LIN {X 0,Y 440.779,Z 670.72,A -85,B 0,C 180,E1 8798.14,E2 8798.14} C_VEL
LIN {X 0,Y 437.985,Z 696.597,A -85,B 0,C 180,E1 8801.691,E2 8801.691} C_VEL
LIN {X 0,Y 435.886,Z 717.468,A -85,B 0,C 180,E1 8805.769,E2 8805.769} C_VEL
LIN {X 0,Y 434.77,Z 732.2,A -85,B 0,C 180,E1 8810.004,E2 8810.004} C_VEL
LIN {X 0,Y 434.32,Z 740.921,A -85,B 0,C 180,E1 8814.015,E2 8814.015} C_VEL
LIN {X 0,Y 434.115,Z 745.167,A -85,B 0,C 180,E1 8818.005,E2 8818.005} C_VEL
LIN {X 0,Y 434.245,Z 745.196,A -85,B 0,C 180,E1 8821.989,E2 8821.989} C_VEL
LIN {X 0,Y 434.323,Z 741.018,A -85,B 0,C 180,E1 8825.98,E2 8825.98} C_VEL
LIN {X 0,Y 434.91,Z 730.868,A -85,B 0,C 180,E1 8830.493,E2 8830.493} C_VEL
LIN {X 0,Y 436.273,Z 714.903,A -85,B 0,C 180,E1 8834.818,E2 8834.818} C_VEL
LIN {X 0,Y 438.333,Z 693.903,A -85,B 0,C 180,E1 8838.674,E2 8838.674} C_VEL
LIN {X 0,Y 441.086,Z 667.612,A -85,B 0,C 180,E1 8842.103,E2 8842.103} C_VEL
LIN {X 0,Y 444.082,Z 637.747,A -85,B 0,C 180,E1 8844.863,E2 8844.863} C_VEL
LIN {X 0,Y 446.927,Z 603.336,A -85,B 0,C 180,E1 8847.021,E2 8847.021} C_VEL
LIN {X 0,Y 448.217,Z 571.069,A -85,B 0,C 180,E1 8848.344,E2 8848.344} C_VEL
LIN {X 0,Y 435.993,Z 537.616,A -85,B 0,C 180,E1 8850.23,E2 8850.23} C_VEL
LIN {X 0,Y 432.921,Z 529.66,A -85,B 0,C 180,E1 8850.787,E2 8850.787} C_VEL
LIN {X 0,Y 432.776,Z 529.66,A -85,B 0,C 180,E1 8856.684,E2 8856.684} C_VEL
LIN {X 0,Y 432.689,Z 529.66,A -85,B 0,C 180,E1 8862.916,E2 8862.916} C_VEL
LIN {X 0,Y 432.797,Z 529.66,A -85,B 0,C 180,E1 8868.514,E2 8868.514} C_VEL
LIN {X 0,Y 432.948,Z 530.172,A -85,B 0,C 180,E1 8874.712,E2 8874.712} C_VEL
LIN {X 0,Y 445.086,Z 561.236,A -85,B 0,C 180,E1 8876.436,E2 8876.436} C_VEL
LIN {X 0,Y 450.898,Z 581.785,A -85,B 0,C 180,E1 8877.342,E2 8877.342} C_VEL
LIN {X 0,Y 450.65,Z 585.781,A -85,B 0,C 180,E1 8877.438,E2 8877.438} C_VEL
LIN {X 0,Y 446.315,Z 602.62,A -85,B 0,C 180,E1 8877.748,E2 8877.748} C_VEL
LIN {X 0,Y 441.689,Z 619.155,A -85,B 0,C 180,E1 8878.204,E2 8878.204} C_VEL
LIN {X 0,Y 438.626,Z 656.172,A -85,B 0,C 180,E1 8880.362,E2 8880.362} C_VEL
LIN {X 0,Y 435.196,Z 690.045,A -85,B 0,C 180,E1 8883.209,E2 8883.209} C_VEL
LIN {X 0,Y 432.003,Z 719.089,A -85,B 0,C 180,E1 8886.59,E2 8886.59} C_VEL
LIN {X 0,Y 429.38,Z 743.866,A -85,B 0,C 180,E1 8890.498,E2 8890.498} C_VEL
LIN {X 0,Y 427.594,Z 764.222,A -85,B 0,C 180,E1 8894.915,E2 8894.915} C_VEL
LIN {X 0,Y 426.692,Z 778.272,A -85,B 0,C 180,E1 8899.301,E2 8899.301} C_VEL
LIN {X 0,Y 426.293,Z 787.499,A -85,B 0,C 180,E1 8903.905,E2 8903.905} C_VEL
LIN {X 0,Y 426.191,Z 791.357,A -85,B 0,C 180,E1 8907.972,E2 8907.972} C_VEL
LIN {X 0,Y 426.311,Z 791.428,A -85,B 0,C 180,E1 8912.029,E2 8912.029} C_VEL
LIN {X 0,Y 426.365,Z 786.444,A -85,B 0,C 180,E1 8916.931,E2 8916.931} C_VEL
LIN {X 0,Y 426.806,Z 776.037,A -85,B 0,C 180,E1 8921.731,E2 8921.731} C_VEL
LIN {X 0,Y 428.059,Z 760.201,A -85,B 0,C 180,E1 8926.381,E2 8926.381} C_VEL
LIN {X 0,Y 430.302,Z 739.014,A -85,B 0,C 180,E1 8930.726,E2 8930.726} C_VEL
LIN {X 0,Y 433.467,Z 712.547,A -85,B 0,C 180,E1 8934.693,E2 8934.693} C_VEL
LIN {X 0,Y 437.226,Z 681.333,A -85,B 0,C 180,E1 8938.103,E2 8938.103} C_VEL
LIN {X 0,Y 440.893,Z 647.439,A -85,B 0,C 180,E1 8940.748,E2 8940.748} C_VEL
LIN {X 0,Y 444.152,Z 610.628,A -85,B 0,C 180,E1 8942.694,E2 8942.694} C_VEL
LIN {X 0,Y 445.424,Z 580.542,A -85,B 0,C 180,E1 8943.715,E2 8943.715} C_VEL
LIN {X 0,Y 424.959,Z 529.66,A -85,B 0,C 180,E1 8946.415,E2 8946.415} C_VEL
LIN {X 0,Y 424.88,Z 529.66,A -85,B 0,C 180,E1 8952.44,E2 8952.44} C_VEL
LIN {X 0,Y 424.897,Z 529.66,A -85,B 0,C 180,E1 8958.229,E2 8958.229} C_VEL
LIN {X 0,Y 424.87,Z 529.66,A -85,B 0,C 180,E1 8964.775,E2 8964.775} C_VEL
LIN {X 0,Y 424.949,Z 529.66,A -85,B 0,C 180,E1 8970.193,E2 8970.193} C_VEL
LIN {X 0,Y 425.265,Z 529.66,A -85,B 0,C 180,E1 8977.307,E2 8977.307} C_VEL
LIN {X 0,Y 425.342,Z 529.66,A -85,B 0,C 180,E1 8983.515,E2 8983.515} C_VEL
LIN {X 0,Y 425.52,Z 529.66,A -85,B 0,C 180,E1 8989.79,E2 8989.79} C_VEL
LIN {X 0,Y 425.85,Z 529.66,A -85,B 0,C 180,E1 8995.939,E2 8995.939} C_VEL
LIN {X 0,Y 425.934,Z 529.66,A -85,B 0,C 180,E1 9002.033,E2 9002.033} C_VEL
LIN {X 0,Y 425.693,Z 529.66,A -85,B 0,C 180,E1 9008.154,E2 9008.154} C_VEL
LIN {X 0,Y 425.526,Z 529.66,A -85,B 0,C 180,E1 9014.376,E2 9014.376} C_VEL
LIN {X 0,Y 425.277,Z 529.66,A -85,B 0,C 180,E1 9020.785,E2 9020.785} C_VEL
LIN {X 0,Y 425.011,Z 529.66,A -85,B 0,C 180,E1 9027.491,E2 9027.491} C_VEL
LIN {X 0,Y 424.899,Z 529.66,A -85,B 0,C 180,E1 9032.192,E2 9032.192} C_VEL
LIN {X 0,Y 424.756,Z 529.66,A -85,B 0,C 180,E1 9038.594,E2 9038.594} C_VEL
LIN {X 0,Y 424.951,Z 529.66,A -85,B 0,C 180,E1 9042.155,E2 9042.155} C_VEL
LIN {X 0,Y 435.694,Z 565.218,A -85,B 0,C 180,E1 9043.418,E2 9043.418} C_VEL
LIN {X 0,Y 434.717,Z 630.818,A -85,B 0,C 180,E1 9044.664,E2 9044.664} C_VEL
LIN {X 0,Y 433.297,Z 660.085,A -85,B 0,C 180,E1 9046.045,E2 9046.045} C_VEL
LIN {X 0,Y 431.378,Z 686.68,A -85,B 0,C 180,E1 9048.181,E2 9048.181} C_VEL
LIN {X 0,Y 429.488,Z 707.938,A -85,B 0,C 180,E1 9050.77,E2 9050.77} C_VEL
LIN {X 0,Y 427.948,Z 726.147,A -85,B 0,C 180,E1 9054.054,E2 9054.054} C_VEL
LIN {X 0,Y 427.035,Z 738.343,A -85,B 0,C 180,E1 9057.427,E2 9057.427} C_VEL
LIN {X 0,Y 426.389,Z 746.323,A -85,B 0,C 180,E1 9061.339,E2 9061.339} C_VEL
LIN {X 0,Y 425.966,Z 748.61,A -85,B 0,C 180,E1 9064.842,E2 9064.842} C_VEL
LIN {X 0,Y 426.245,Z 746.682,A -85,B 0,C 180,E1 9068.177,E2 9068.177} C_VEL
LIN {X 0,Y 426.915,Z 739.239,A -85,B 0,C 180,E1 9072.082,E2 9072.082} C_VEL
LIN {X 0,Y 427.894,Z 726.465,A -85,B 0,C 180,E1 9075.707,E2 9075.707} C_VEL
LIN {X 0,Y 429.374,Z 708.345,A -85,B 0,C 180,E1 9079.001,E2 9079.001} C_VEL
LIN {X 0,Y 431.265,Z 686.257,A -85,B 0,C 180,E1 9081.7,E2 9081.7} C_VEL
LIN {X 0,Y 433.143,Z 660.725,A -85,B 0,C 180,E1 9083.761,E2 9083.761} C_VEL
LIN {X 0,Y 434.519,Z 631.681,A -85,B 0,C 180,E1 9085.163,E2 9085.163} C_VEL
LIN {X 0,Y 435.3,Z 581.985,A -85,B 0,C 180,E1 9086.161,E2 9086.161} C_VEL
LIN {X 0,Y 434.75,Z 560.582,A -85,B 0,C 180,E1 9086.562,E2 9086.562} C_VEL
LIN {X 0,Y 425.9,Z 529.66,A -85,B 0,C 180,E1 9087.611,E2 9087.611} C_VEL
LIN {X 0,Y 425.874,Z 529.66,A -85,B 0,C 180,E1 9094.063,E2 9094.063} C_VEL
LIN {X 0,Y 425.568,Z 529.66,A -85,B 0,C 180,E1 9100.211,E2 9100.211} C_VEL
LIN {X 0,Y 425.337,Z 529.66,A -85,B 0,C 180,E1 9106.679,E2 9106.679} C_VEL
LIN {X 0,Y 425.185,Z 529.66,A -85,B 0,C 180,E1 9112.978,E2 9112.978} C_VEL
LIN {X 0,Y 424.896,Z 529.66,A -85,B 0,C 180,E1 9119.814,E2 9119.814} C_VEL
LIN {X 0,Y 424.929,Z 529.66,A -85,B 0,C 180,E1 9127.134,E2 9127.134} C_VEL
LIN {X 0,Y 424.896,Z 529.66,A -85,B 0,C 180,E1 9132.435,E2 9132.435} C_VEL
LIN {X 0,Y 424.889,Z 529.66,A -85,B 0,C 180,E1 9138.228,E2 9138.228} C_VEL
LIN {X 0,Y 424.827,Z 529.66,A -85,B 0,C 180,E1 9144.78,E2 9144.78} C_VEL
LIN {X 0,Y 424.953,Z 529.734,A -85,B 0,C 180,E1 9148.889,E2 9148.889} C_VEL
LIN {X 0,Y 441.951,Z 574.346,A -85,B 0,C 180,E1 9151.179,E2 9151.179} C_VEL
LIN {X 0,Y 439.632,Z 608.94,A -85,B 0,C 180,E1 9152.658,E2 9152.658} C_VEL
LIN {X 0,Y 436.632,Z 641.055,A -85,B 0,C 180,E1 9154.843,E2 9154.843} C_VEL
LIN {X 0,Y 433.349,Z 670.624,A -85,B 0,C 180,E1 9157.745,E2 9157.745} C_VEL
LIN {X 0,Y 430.36,Z 696.708,A -85,B 0,C 180,E1 9161.364,E2 9161.364} C_VEL
LIN {X 0,Y 428.173,Z 717.656,A -85,B 0,C 180,E1 9165.507,E2 9165.507} C_VEL
LIN {X 0,Y 426.916,Z 732.492,A -85,B 0,C 180,E1 9169.818,E2 9169.818} C_VEL
LIN {X 0,Y 426.442,Z 741.289,A -85,B 0,C 180,E1 9173.904,E2 9173.904} C_VEL
LIN {X 0,Y 426.226,Z 745.581,A -85,B 0,C 180,E1 9177.968,E2 9177.968} C_VEL
LIN {X 0,Y 426.354,Z 745.626,A -85,B 0,C 180,E1 9182.026,E2 9182.026} C_VEL
LIN {X 0,Y 426.449,Z 741.433,A -85,B 0,C 180,E1 9186.091,E2 9186.091} C_VEL
LIN {X 0,Y 427.089,Z 731.223,A -85,B 0,C 180,E1 9190.687,E2 9190.687} C_VEL
LIN {X 0,Y 428.485,Z 715.836,A -85,B 0,C 180,E1 9194.938,E2 9194.938} C_VEL
LIN {X 0,Y 430.681,Z 694.719,A -85,B 0,C 180,E1 9198.917,E2 9198.917} C_VEL
LIN {X 0,Y 433.568,Z 668.876,A -85,B 0,C 180,E1 9202.372,E2 9202.372} C_VEL
LIN {X 0,Y 436.698,Z 639.491,A -85,B 0,C 180,E1 9205.166,E2 9205.166} C_VEL
LIN {X 0,Y 439.719,Z 605.426,A -85,B 0,C 180,E1 9207.386,E2 9207.386} C_VEL
LIN {X 0,Y 441.347,Z 573.368,A -85,B 0,C 180,E1 9208.771,E2 9208.771} C_VEL
LIN {X 0,Y 430.113,Z 541.822,A -85,B 0,C 180,E1 9210.654,E2 9210.654} C_VEL
LIN {X 0,Y 424.97,Z 529.66,A -85,B 0,C 180,E1 9211.55,E2 9211.55} C_VEL
LIN {X 0,Y 424.803,Z 529.66,A -85,B 0,C 180,E1 9218.605,E2 9218.605} C_VEL
LIN {X 0,Y 424.845,Z 529.66,A -85,B 0,C 180,E1 9225.261,E2 9225.261} C_VEL
LIN {X 0,Y 424.886,Z 529.66,A -85,B 0,C 180,E1 9231.378,E2 9231.378} C_VEL
LIN {X 0,Y 424.949,Z 529.66,A -85,B 0,C 180,E1 9233.886,E2 9233.886} C_VEL
LIN {X 0,Y 437.607,Z 560.962,A -85,B 0,C 180,E1 9235.846,E2 9235.846} C_VEL
LIN {X 0,Y 443.854,Z 583.141,A -85,B 0,C 180,E1 9236.892,E2 9236.892} C_VEL
LIN {X 0,Y 441.689,Z 619.155,A -85,B 0,C 180,E1 9238.204,E2 9238.204} C_VEL
LIN {X 0,Y 436.799,Z 635.43,A -85,B 0,C 180,E1 9238.792,E2 9238.792} C_VEL
LIN {X 0,Y 431.895,Z 651.113,A -85,B 0,C 180,E1 9239.573,E2 9239.573} C_VEL
LIN {X 0,Y 428.172,Z 685.606,A -85,B 0,C 180,E1 9242.404,E2 9242.404} C_VEL
LIN {X 0,Y 424.762,Z 716.142,A -85,B 0,C 180,E1 9245.888,E2 9245.888} C_VEL
LIN {X 0,Y 421.934,Z 741.599,A -85,B 0,C 180,E1 9249.866,E2 9249.866} C_VEL
LIN {X 0,Y 419.958,Z 761.432,A -85,B 0,C 180,E1 9254.1,E2 9254.1} C_VEL
LIN {X 0,Y 418.851,Z 776.255,A -85,B 0,C 180,E1 9258.572,E2 9258.572} C_VEL
LIN {X 0,Y 418.521,Z 785.886,A -85,B 0,C 180,E1 9263.074,E2 9263.074} C_VEL
LIN {X 0,Y 418.302,Z 790.915,A -85,B 0,C 180,E1 9267.934,E2 9267.934} C_VEL
LIN {X 0,Y 418.414,Z 791.006,A -85,B 0,C 180,E1 9272.068,E2 9272.068} C_VEL
LIN {X 0,Y 418.482,Z 786.232,A -85,B 0,C 180,E1 9276.916,E2 9276.916} C_VEL
LIN {X 0,Y 418.867,Z 776.93,A -85,B 0,C 180,E1 9281.429,E2 9281.429} C_VEL
LIN {X 0,Y 420.103,Z 761.642,A -85,B 0,C 180,E1 9286.164,E2 9286.164} C_VEL
LIN {X 0,Y 422.364,Z 740.864,A -85,B 0,C 180,E1 9290.66,E2 9290.66} C_VEL
LIN {X 0,Y 425.533,Z 715.539,A -85,B 0,C 180,E1 9294.625,E2 9294.625} C_VEL
LIN {X 0,Y 429.177,Z 686.549,A -85,B 0,C 180,E1 9297.99,E2 9297.99} C_VEL
LIN {X 0,Y 433.086,Z 653.405,A -85,B 0,C 180,E1 9300.782,E2 9300.782} C_VEL
LIN {X 0,Y 436.604,Z 616.909,A -85,B 0,C 180,E1 9302.874,E2 9302.874} C_VEL
LIN {X 0,Y 438.552,Z 583.038,A -85,B 0,C 180,E1 9304.117,E2 9304.117} C_VEL
LIN {X 0,Y 417.895,Z 533.217,A -85,B 0,C 180,E1 9306.828,E2 9306.828} C_VEL
LIN {X 0,Y 417.028,Z 529.66,A -85,B 0,C 180,E1 9307.085,E2 9307.085} C_VEL
LIN {X 0,Y 416.896,Z 529.66,A -85,B 0,C 180,E1 9313.626,E2 9313.626} C_VEL
LIN {X 0,Y 416.928,Z 529.66,A -85,B 0,C 180,E1 9319.47,E2 9319.47} C_VEL
LIN {X 0,Y 416.956,Z 529.66,A -85,B 0,C 180,E1 9324.62,E2 9324.62} C_VEL
LIN {X 0,Y 417.055,Z 529.66,A -85,B 0,C 180,E1 9331.945,E2 9331.945} C_VEL
LIN {X 0,Y 417.359,Z 529.66,A -85,B 0,C 180,E1 9338.807,E2 9338.807} C_VEL
LIN {X 0,Y 417.431,Z 529.66,A -85,B 0,C 180,E1 9345.345,E2 9345.345} C_VEL
LIN {X 0,Y 417.745,Z 529.66,A -85,B 0,C 180,E1 9351.695,E2 9351.695} C_VEL
LIN {X 0,Y 418.188,Z 529.66,A -85,B 0,C 180,E1 9357.935,E2 9357.935} C_VEL
LIN {X 0,Y 417.998,Z 529.66,A -85,B 0,C 180,E1 9364.143,E2 9364.143} C_VEL
LIN {X 0,Y 417.696,Z 529.66,A -85,B 0,C 180,E1 9370.409,E2 9370.409} C_VEL
LIN {X 0,Y 417.505,Z 529.66,A -85,B 0,C 180,E1 9376.809,E2 9376.809} C_VEL
LIN {X 0,Y 417.223,Z 529.66,A -85,B 0,C 180,E1 9383.446,E2 9383.446} C_VEL
LIN {X 0,Y 417.009,Z 529.66,A -85,B 0,C 180,E1 9390.441,E2 9390.441} C_VEL
LIN {X 0,Y 416.884,Z 529.66,A -85,B 0,C 180,E1 9397.217,E2 9397.217} C_VEL
LIN {X 0,Y 417.033,Z 530.044,A -85,B 0,C 180,E1 9401.713,E2 9401.713} C_VEL
LIN {X 0,Y 428.371,Z 565.36,A -85,B 0,C 180,E1 9403.023,E2 9403.023} C_VEL
LIN {X 0,Y 427.349,Z 630.6,A -85,B 0,C 180,E1 9404.273,E2 9404.273} C_VEL
LIN {X 0,Y 425.884,Z 659.666,A -85,B 0,C 180,E1 9405.646,E2 9405.646} C_VEL
LIN {X 0,Y 423.939,Z 686.175,A -85,B 0,C 180,E1 9407.781,E2 9407.781} C_VEL
LIN {X 0,Y 421.85,Z 708.373,A -85,B 0,C 180,E1 9410.512,E2 9410.512} C_VEL
LIN {X 0,Y 420.196,Z 726.411,A -85,B 0,C 180,E1 9413.818,E2 9413.818} C_VEL
LIN {X 0,Y 419.207,Z 738.84,A -85,B 0,C 180,E1 9417.319,E2 9417.319} C_VEL
LIN {X 0,Y 418.572,Z 746.3,A -85,B 0,C 180,E1 9420.963,E2 9420.963} C_VEL
LIN {X 0,Y 418.098,Z 748.939,A -85,B 0,C 180,E1 9424.466,E2 9424.466} C_VEL
LIN {X 0,Y 418.274,Z 747.576,A -85,B 0,C 180,E1 9427.785,E2 9427.785} C_VEL
LIN {X 0,Y 418.967,Z 740.983,A -85,B 0,C 180,E1 9431.666,E2 9431.666} C_VEL
LIN {X 0,Y 419.942,Z 728.806,A -85,B 0,C 180,E1 9435.431,E2 9435.431} C_VEL
LIN {X 0,Y 421.432,Z 711.577,A -85,B 0,C 180,E1 9438.813,E2 9438.813} C_VEL
LIN {X 0,Y 423.397,Z 689.707,A -85,B 0,C 180,E1 9441.674,E2 9441.674} C_VEL
LIN {X 0,Y 425.454,Z 664.112,A -85,B 0,C 180,E1 9443.891,E2 9443.891} C_VEL
LIN {X 0,Y 426.937,Z 636.104,A -85,B 0,C 180,E1 9445.374,E2 9445.374} C_VEL
LIN {X 0,Y 427.685,Z 601.221,A -85,B 0,C 180,E1 9446.21,E2 9446.21} C_VEL
LIN {X 0,Y 427.664,Z 562.945,A -85,B 0,C 180,E1 9446.892,E2 9446.892} C_VEL
LIN {X 0,Y 418.027,Z 529.66,A -85,B 0,C 180,E1 9448.06,E2 9448.06} C_VEL
LIN {X 0,Y 417.962,Z 529.66,A -85,B 0,C 180,E1 9454.14,E2 9454.14} C_VEL
LIN {X 0,Y 417.64,Z 529.66,A -85,B 0,C 180,E1 9460.407,E2 9460.407} C_VEL
LIN {X 0,Y 417.436,Z 529.66,A -85,B 0,C 180,E1 9466.809,E2 9466.809} C_VEL
LIN {X 0,Y 417.211,Z 529.66,A -85,B 0,C 180,E1 9473.443,E2 9473.443} C_VEL
LIN {X 0,Y 416.983,Z 529.66,A -85,B 0,C 180,E1 9480.439,E2 9480.439} C_VEL
LIN {X 0,Y 417.002,Z 529.66,A -85,B 0,C 180,E1 9487.963,E2 9487.963} C_VEL
LIN {X 0,Y 416.909,Z 529.66,A -85,B 0,C 180,E1 9493.62,E2 9493.62} C_VEL
LIN {X 0,Y 416.931,Z 529.66,A -85,B 0,C 180,E1 9499.467,E2 9499.467} C_VEL
LIN {X 0,Y 416.912,Z 529.66,A -85,B 0,C 180,E1 9504.609,E2 9504.609} C_VEL
LIN {X 0,Y 416.996,Z 529.66,A -85,B 0,C 180,E1 9508.266,E2 9508.266} C_VEL
LIN {X 0,Y 434.727,Z 576.141,A -85,B 0,C 180,E1 9510.767,E2 9510.767} C_VEL
LIN {X 0,Y 432.337,Z 610.732,A -85,B 0,C 180,E1 9512.31,E2 9512.31} C_VEL
LIN {X 0,Y 429.174,Z 642.858,A -85,B 0,C 180,E1 9514.571,E2 9514.571} C_VEL
LIN {X 0,Y 425.668,Z 672.623,A -85,B 0,C 180,E1 9517.596,E2 9517.596} C_VEL
LIN {X 0,Y 422.619,Z 698.114,A -85,B 0,C 180,E1 9521.253,E2 9521.253} C_VEL
LIN {X 0,Y 420.361,Z 718.702,A -85,B 0,C 180,E1 9525.444,E2 9525.444} C_VEL
LIN {X 0,Y 419.092,Z 732.779,A -85,B 0,C 180,E1 9529.626,E2 9529.626} C_VEL
LIN {X 0,Y 418.567,Z 741.645,A -85,B 0,C 180,E1 9533.788,E2 9533.788} C_VEL
LIN {X 0,Y 418.337,Z 745.987,A -85,B 0,C 180,E1 9537.93,E2 9537.93} C_VEL
LIN {X 0,Y 418.463,Z 746.055,A -85,B 0,C 180,E1 9542.064,E2 9542.064} C_VEL
LIN {X 0,Y 418.578,Z 741.854,A -85,B 0,C 180,E1 9546.206,E2 9546.206} C_VEL
LIN {X 0,Y 419.291,Z 731.598,A -85,B 0,C 180,E1 9550.888,E2 9550.888} C_VEL
LIN {X 0,Y 420.855,Z 715.69,A -85,B 0,C 180,E1 9555.33,E2 9555.33} C_VEL
LIN {X 0,Y 423.128,Z 694.983,A -85,B 0,C 180,E1 9559.268,E2 9559.268} C_VEL
LIN {X 0,Y 426.258,Z 668.558,A -85,B 0,C 180,E1 9562.84,E2 9562.84} C_VEL
LIN {X 0,Y 429.692,Z 638.009,A -85,B 0,C 180,E1 9565.755,E2 9565.755} C_VEL
LIN {X 0,Y 432.961,Z 603.471,A -85,B 0,C 180,E1 9567.993,E2 9567.993} C_VEL
LIN {X 0,Y 434.361,Z 575.23,A -85,B 0,C 180,E1 9569.244,E2 9569.244} C_VEL
LIN {X 0,Y 423.803,Z 544.782,A -85,B 0,C 180,E1 9571.19,E2 9571.19} C_VEL
LIN {X 0,Y 416.971,Z 529.66,A -85,B 0,C 180,E1 9572.574,E2 9572.574} C_VEL
LIN {X 0,Y 416.915,Z 529.66,A -85,B 0,C 180,E1 9577.97,E2 9577.97} C_VEL
LIN {X 0,Y 416.821,Z 529.66,A -85,B 0,C 180,E1 9583.612,E2 9583.612} C_VEL
LIN {X 0,Y 416.919,Z 529.66,A -85,B 0,C 180,E1 9589.465,E2 9589.465} C_VEL
LIN {X 0,Y 417.015,Z 529.66,A -85,B 0,C 180,E1 9592.993,E2 9592.993} C_VEL
LIN {X 0,Y 429.677,Z 559.319,A -85,B 0,C 180,E1 9595.129,E2 9595.129} C_VEL
LIN {X 0,Y 436.844,Z 585.679,A -85,B 0,C 180,E1 9596.449,E2 9596.449} C_VEL
LIN {X 0,Y 434.25,Z 623.659,A -85,B 0,C 180,E1 9597.953,E2 9597.953} C_VEL
LIN {X 0,Y 431.895,Z 651.113,A -85,B 0,C 180,E1 9599.573,E2 9599.573} C_VEL
LIN {X 0,Y 426.638,Z 666.431,A -85,B 0,C 180,E1 9600.487,E2 9600.487} C_VEL
LIN {X 0,Y 421.629,Z 679.32,A -85,B 0,C 180,E1 9601.391,E2 9601.391} C_VEL
LIN {X 0,Y 421.361,Z 681.101,A -85,B 0,C 180,E1 9601.56,E2 9601.56} C_VEL
LIN {X 0,Y 417.624,Z 712.349,A -85,B 0,C 180,E1 9605.061,E2 9605.061} C_VEL
LIN {X 0,Y 414.428,Z 739.351,A -85,B 0,C 180,E1 9609.207,E2 9609.207} C_VEL
LIN {X 0,Y 412.187,Z 760.753,A -85,B 0,C 180,E1 9613.792,E2 9613.792} C_VEL
LIN {X 0,Y 411.008,Z 775.683,A -85,B 0,C 180,E1 9618.351,E2 9618.351} C_VEL
LIN {X 0,Y 410.634,Z 785.181,A -85,B 0,C 180,E1 9622.807,E2 9622.807} C_VEL
LIN {X 0,Y 410.409,Z 790.48,A -85,B 0,C 180,E1 9627.894,E2 9627.894} C_VEL
LIN {X 0,Y 410.518,Z 790.584,A -85,B 0,C 180,E1 9632.107,E2 9632.107} C_VEL
LIN {X 0,Y 410.595,Z 785.632,A -85,B 0,C 180,E1 9637.15,E2 9637.15} C_VEL
LIN {X 0,Y 411.019,Z 776.422,A -85,B 0,C 180,E1 9641.65,E2 9641.65} C_VEL
LIN {X 0,Y 412.313,Z 761.034,A -85,B 0,C 180,E1 9646.478,E2 9646.478} C_VEL
LIN {X 0,Y 414.742,Z 740.055,A -85,B 0,C 180,E1 9651.058,E2 9651.058} C_VEL
LIN {X 0,Y 418.098,Z 714.515,A -85,B 0,C 180,E1 9655.093,E2 9655.093} C_VEL
LIN {X 0,Y 422.065,Z 684.463,A -85,B 0,C 180,E1 9658.589,E2 9658.589} C_VEL
LIN {X 0,Y 426.071,Z 651.539,A -85,B 0,C 180,E1 9661.345,E2 9661.345} C_VEL
LIN {X 0,Y 429.646,Z 615.789,A -85,B 0,C 180,E1 9663.394,E2 9663.394} C_VEL
LIN {X 0,Y 431.283,Z 584.466,A -85,B 0,C 180,E1 9664.586,E2 9664.586} C_VEL
LIN {X 0,Y 410.251,Z 533.741,A -85,B 0,C 180,E1 9667.433,E2 9667.433} C_VEL
LIN {X 0,Y 409.116,Z 529.66,A -85,B 0,C 180,E1 9667.756,E2 9667.756} C_VEL
LIN {X 0,Y 408.9,Z 529.66,A -85,B 0,C 180,E1 9674.522,E2 9674.522} C_VEL
LIN {X 0,Y 408.973,Z 529.66,A -85,B 0,C 180,E1 9681.157,E2 9681.157} C_VEL
LIN {X 0,Y 408.999,Z 529.66,A -85,B 0,C 180,E1 9688.059,E2 9688.059} C_VEL
LIN {X 0,Y 409.188,Z 529.66,A -85,B 0,C 180,E1 9693.738,E2 9693.738} C_VEL
LIN {X 0,Y 409.471,Z 529.66,A -85,B 0,C 180,E1 9700.633,E2 9700.633} C_VEL
LIN {X 0,Y 409.632,Z 529.66,A -85,B 0,C 180,E1 9707.234,E2 9707.234} C_VEL
LIN {X 0,Y 409.989,Z 529.66,A -85,B 0,C 180,E1 9713.664,E2 9713.664} C_VEL
LIN {X 0,Y 410.217,Z 529.66,A -85,B 0,C 180,E1 9720.003,E2 9720.003} C_VEL
LIN {X 0,Y 409.962,Z 529.66,A -85,B 0,C 180,E1 9726.367,E2 9726.367} C_VEL
LIN {X 0,Y 409.75,Z 529.66,A -85,B 0,C 180,E1 9732.768,E2 9732.768} C_VEL
LIN {X 0,Y 409.472,Z 529.66,A -85,B 0,C 180,E1 9739.373,E2 9739.373} C_VEL
LIN {X 0,Y 409.148,Z 529.66,A -85,B 0,C 180,E1 9746.271,E2 9746.271} C_VEL
LIN {X 0,Y 408.99,Z 529.66,A -85,B 0,C 180,E1 9753.606,E2 9753.606} C_VEL
LIN {X 0,Y 409.032,Z 529.66,A -85,B 0,C 180,E1 9761.19,E2 9761.19} C_VEL
LIN {X 0,Y 421.102,Z 567.522,A -85,B 0,C 180,E1 9762.651,E2 9762.651} C_VEL
LIN {X 0,Y 419.981,Z 631.434,A -85,B 0,C 180,E1 9763.905,E2 9763.905} C_VEL
LIN {X 0,Y 418.415,Z 660.793,A -85,B 0,C 180,E1 9765.333,E2 9765.333} C_VEL
LIN {X 0,Y 416.45,Z 686.36,A -85,B 0,C 180,E1 9767.436,E2 9767.436} C_VEL
LIN {X 0,Y 414.282,Z 707.88,A -85,B 0,C 180,E1 9770.096,E2 9770.096} C_VEL
LIN {X 0,Y 412.565,Z 724.992,A -85,B 0,C 180,E1 9773.188,E2 9773.188} C_VEL
LIN {X 0,Y 411.382,Z 739.144,A -85,B 0,C 180,E1 9777.138,E2 9777.138} C_VEL
LIN {X 0,Y 410.773,Z 746.003,A -85,B 0,C 180,E1 9780.402,E2 9780.402} C_VEL
LIN {X 0,Y 410.229,Z 749.179,A -85,B 0,C 180,E1 9783.805,E2 9783.805} C_VEL
LIN {X 0,Y 410.258,Z 748.749,A -85,B 0,C 180,E1 9786.864,E2 9786.864} C_VEL
LIN {X 0,Y 410.908,Z 743.746,A -85,B 0,C 180,E1 9790.699,E2 9790.699} C_VEL
LIN {X 0,Y 411.758,Z 733.098,A -85,B 0,C 180,E1 9794.591,E2 9794.591} C_VEL
LIN {X 0,Y 413.176,Z 717.285,A -85,B 0,C 180,E1 9798.144,E2 9798.144} C_VEL
LIN {X 0,Y 415.261,Z 696.144,A -85,B 0,C 180,E1 9801.282,E2 9801.282} C_VEL
LIN {X 0,Y 417.472,Z 670.681,A -85,B 0,C 180,E1 9803.774,E2 9803.774} C_VEL
LIN {X 0,Y 419.237,Z 642.542,A -85,B 0,C 180,E1 9805.483,E2 9805.483} C_VEL
LIN {X 0,Y 420.191,Z 612.074,A -85,B 0,C 180,E1 9806.403,E2 9806.403} C_VEL
LIN {X 0,Y 420.002,Z 563.43,A -85,B 0,C 180,E1 9807.297,E2 9807.297} C_VEL
LIN {X 0,Y 410.114,Z 529.66,A -85,B 0,C 180,E1 9808.55,E2 9808.55} C_VEL
LIN {X 0,Y 410.051,Z 529.66,A -85,B 0,C 180,E1 9814.22,E2 9814.22} C_VEL
LIN {X 0,Y 409.735,Z 529.66,A -85,B 0,C 180,E1 9820.61,E2 9820.61} C_VEL
LIN {X 0,Y 409.515,Z 529.66,A -85,B 0,C 180,E1 9827.144,E2 9827.144} C_VEL
LIN {X 0,Y 409.267,Z 529.66,A -85,B 0,C 180,E1 9833.926,E2 9833.926} C_VEL
LIN {X 0,Y 408.989,Z 529.66,A -85,B 0,C 180,E1 9841.099,E2 9841.099} C_VEL
LIN {X 0,Y 409.054,Z 529.66,A -85,B 0,C 180,E1 9846.173,E2 9846.173} C_VEL
LIN {X 0,Y 408.913,Z 529.66,A -85,B 0,C 180,E1 9852.431,E2 9852.431} C_VEL
LIN {X 0,Y 408.905,Z 529.66,A -85,B 0,C 180,E1 9858.371,E2 9858.371} C_VEL
LIN {X 0,Y 409.005,Z 529.66,A -85,B 0,C 180,E1 9864.258,E2 9864.258} C_VEL
LIN {X 0,Y 409.027,Z 529.66,A -85,B 0,C 180,E1 9867.661,E2 9867.661} C_VEL
LIN {X 0,Y 427.216,Z 577.131,A -85,B 0,C 180,E1 9870.294,E2 9870.294} C_VEL
LIN {X 0,Y 425.045,Z 612.306,A -85,B 0,C 180,E1 9871.948,E2 9871.948} C_VEL
LIN {X 0,Y 421.735,Z 644.204,A -85,B 0,C 180,E1 9874.255,E2 9874.255} C_VEL
LIN {X 0,Y 418.147,Z 673.226,A -85,B 0,C 180,E1 9877.277,E2 9877.277} C_VEL
LIN {X 0,Y 414.946,Z 698.687,A -85,B 0,C 180,E1 9880.996,E2 9880.996} C_VEL
LIN {X 0,Y 412.625,Z 718.862,A -85,B 0,C 180,E1 9885.165,E2 9885.165} C_VEL
LIN {X 0,Y 411.255,Z 733.056,A -85,B 0,C 180,E1 9889.426,E2 9889.426} C_VEL
LIN {X 0,Y 410.696,Z 742.002,A -85,B 0,C 180,E1 9893.669,E2 9893.669} C_VEL
LIN {X 0,Y 410.447,Z 746.397,A -85,B 0,C 180,E1 9897.89,E2 9897.89} C_VEL
LIN {X 0,Y 410.572,Z 746.488,A -85,B 0,C 180,E1 9902.103,E2 9902.103} C_VEL
LIN {X 0,Y 410.712,Z 742.287,A -85,B 0,C 180,E1 9906.325,E2 9906.325} C_VEL
LIN {X 0,Y 411.492,Z 732.007,A -85,B 0,C 180,E1 9911.097,E2 9911.097} C_VEL
LIN {X 0,Y 413.184,Z 716.064,A -85,B 0,C 180,E1 9915.622,E2 9915.622} C_VEL
LIN {X 0,Y 415.558,Z 695.704,A -85,B 0,C 180,E1 9919.568,E2 9919.568} C_VEL
LIN {X 0,Y 418.853,Z 669.539,A -85,B 0,C 180,E1 9923.189,E2 9923.189} C_VEL
LIN {X 0,Y 422.525,Z 638.971,A -85,B 0,C 180,E1 9926.178,E2 9926.178} C_VEL
LIN {X 0,Y 425.931,Z 605.267,A -85,B 0,C 180,E1 9928.429,E2 9928.429} C_VEL
LIN {X 0,Y 427.57,Z 577.368,A -85,B 0,C 180,E1 9929.726,E2 9929.726} C_VEL
LIN {X 0,Y 417.88,Z 548.512,A -85,B 0,C 180,E1 9931.697,E2 9931.697} C_VEL
LIN {X 0,Y 409.013,Z 529.66,A -85,B 0,C 180,E1 9933.597,E2 9933.597} C_VEL
LIN {X 0,Y 408.878,Z 529.66,A -85,B 0,C 180,E1 9939.195,E2 9939.195} C_VEL
LIN {X 0,Y 408.86,Z 529.66,A -85,B 0,C 180,E1 9945.475,E2 9945.475} C_VEL
LIN {X 0,Y 409.138,Z 530.434,A -85,B 0,C 180,E1 9952.017,E2 9952.017} C_VEL
LIN {X 0,Y 421.261,Z 556.41,A -85,B 0,C 180,E1 9954.251,E2 9954.251} C_VEL
LIN {X 0,Y 430.013,Z 586.559,A -85,B 0,C 180,E1 9955.935,E2 9955.935} C_VEL
LIN {X 0,Y 427.079,Z 625.757,A -85,B 0,C 180,E1 9957.565,E2 9957.565} C_VEL
LIN {X 0,Y 423.486,Z 662.422,A -85,B 0,C 180,E1 9959.95,E2 9959.95} C_VEL
LIN {X 0,Y 421.361,Z 681.101,A -85,B 0,C 180,E1 9961.56,E2 9961.56} C_VEL
LIN {X 0,Y 419.427,Z 688.282,A -85,B 0,C 180,E1 9962.209,E2 9962.209} C_VEL
LIN {X 0,Y 410.899,Z 706.88,A -85,B 0,C 180,E1 9963.985,E2 9963.985} C_VEL
LIN {X 0,Y 410.604,Z 708.482,A -85,B 0,C 180,E1 9964.19,E2 9964.19} C_VEL
LIN {X 0,Y 407.128,Z 735.446,A -85,B 0,C 180,E1 9968.246,E2 9968.246} C_VEL
LIN {X 0,Y 404.592,Z 757.994,A -85,B 0,C 180,E1 9972.921,E2 9972.921} C_VEL
LIN {X 0,Y 403.282,Z 773.69,A -85,B 0,C 180,E1 9977.576,E2 9977.576} C_VEL
LIN {X 0,Y 402.742,Z 783.686,A -85,B 0,C 180,E1 9982.024,E2 9982.024} C_VEL
LIN {X 0,Y 402.611,Z 788.528,A -85,B 0,C 180,E1 9985.702,E2 9985.702} C_VEL
LIN {X 0,Y 402.58,Z 790.636,A -85,B 0,C 180,E1 9990.001,E2 9990.001} C_VEL
LIN {X 0,Y 402.607,Z 788.757,A -85,B 0,C 180,E1 9994.3,E2 9994.3} C_VEL
LIN {X 0,Y 402.848,Z 781.975,A -85,B 0,C 180,E1 9999.161,E2 9999.161} C_VEL
LIN {X 0,Y 403.605,Z 769.553,A -85,B 0,C 180,E1 10004.155,E2 10004.155} C_VEL
LIN {X 0,Y 405.514,Z 751.325,A -85,B 0,C 180,E1 10008.994,E2 10008.994} C_VEL
LIN {X 0,Y 408.621,Z 727.865,A -85,B 0,C 180,E1 10013.436,E2 10013.436} C_VEL
LIN {X 0,Y 412.605,Z 699.495,A -85,B 0,C 180,E1 10017.352,E2 10017.352} C_VEL
LIN {X 0,Y 416.979,Z 667.044,A -85,B 0,C 180,E1 10020.583,E2 10020.583} C_VEL
LIN {X 0,Y 421.123,Z 631.828,A -85,B 0,C 180,E1 10023.048,E2 10023.048} C_VEL
LIN {X 0,Y 424.282,Z 595.664,A -85,B 0,C 180,E1 10024.685,E2 10024.685} C_VEL
LIN {X 0,Y 424.006,Z 585.855,A -85,B 0,C 180,E1 10025.066,E2 10025.066} C_VEL
LIN {X 0,Y 402.27,Z 533.657,A -85,B 0,C 180,E1 10028.095,E2 10028.095} C_VEL
LIN {X 0,Y 401.148,Z 529.66,A -85,B 0,C 180,E1 10028.347,E2 10028.347} C_VEL
LIN {X 0,Y 400.993,Z 529.66,A -85,B 0,C 180,E1 10035.644,E2 10035.644} C_VEL
LIN {X 0,Y 401.024,Z 529.66,A -85,B 0,C 180,E1 10042.987,E2 10042.987} C_VEL
LIN {X 0,Y 401.089,Z 529.66,A -85,B 0,C 180,E1 10049.92,E2 10049.92} C_VEL
LIN {X 0,Y 401.321,Z 529.66,A -85,B 0,C 180,E1 10055.572,E2 10055.572} C_VEL
LIN {X 0,Y 401.565,Z 529.66,A -85,B 0,C 180,E1 10062.508,E2 10062.508} C_VEL
LIN {X 0,Y 401.755,Z 529.66,A -85,B 0,C 180,E1 10069.179,E2 10069.179} C_VEL
LIN {X 0,Y 402.134,Z 529.66,A -85,B 0,C 180,E1 10075.699,E2 10075.699} C_VEL
LIN {X 0,Y 402.257,Z 529.66,A -85,B 0,C 180,E1 10082.153,E2 10082.153} C_VEL
LIN {X 0,Y 401.916,Z 529.66,A -85,B 0,C 180,E1 10088.64,E2 10088.64} C_VEL
LIN {X 0,Y 401.733,Z 529.66,A -85,B 0,C 180,E1 10095.247,E2 10095.247} C_VEL
LIN {X 0,Y 401.429,Z 529.66,A -85,B 0,C 180,E1 10102.083,E2 10102.083} C_VEL
LIN {X 0,Y 401.097,Z 529.66,A -85,B 0,C 180,E1 10109.283,E2 10109.283} C_VEL
LIN {X 0,Y 401.021,Z 529.66,A -85,B 0,C 180,E1 10114.366,E2 10114.366} C_VEL
LIN {X 0,Y 401.127,Z 530.404,A -85,B 0,C 180,E1 10120.7,E2 10120.7} C_VEL
LIN {X 0,Y 413.824,Z 568.555,A -85,B 0,C 180,E1 10122.242,E2 10122.242} C_VEL
LIN {X 0,Y 412.655,Z 631.986,A -85,B 0,C 180,E1 10123.514,E2 10123.514} C_VEL
LIN {X 0,Y 411.057,Z 659.991,A -85,B 0,C 180,E1 10124.88,E2 10124.88} C_VEL
LIN {X 0,Y 408.932,Z 686.955,A -85,B 0,C 180,E1 10127.12,E2 10127.12} C_VEL
LIN {X 0,Y 406.528,Z 709.304,A -85,B 0,C 180,E1 10129.968,E2 10129.968} C_VEL
LIN {X 0,Y 404.656,Z 727.177,A -85,B 0,C 180,E1 10133.368,E2 10133.368} C_VEL
LIN {X 0,Y 403.493,Z 740.242,A -85,B 0,C 180,E1 10137.239,E2 10137.239} C_VEL
LIN {X 0,Y 402.803,Z 747.161,A -85,B 0,C 180,E1 10140.855,E2 10140.855} C_VEL
LIN {X 0,Y 402.298,Z 749.679,A -85,B 0,C 180,E1 10144.193,E2 10144.193} C_VEL
LIN {X 0,Y 402.498,Z 748.239,A -85,B 0,C 180,E1 10147.98,E2 10147.98} C_VEL
LIN {X 0,Y 403.298,Z 741.02,A -85,B 0,C 180,E1 10152.21,E2 10152.21} C_VEL
LIN {X 0,Y 404.471,Z 728.362,A -85,B 0,C 180,E1 10156.124,E2 10156.124} C_VEL
LIN {X 0,Y 406.246,Z 710.101,A -85,B 0,C 180,E1 10159.681,E2 10159.681} C_VEL
LIN {X 0,Y 408.528,Z 687.831,A -85,B 0,C 180,E1 10162.571,E2 10162.571} C_VEL
LIN {X 0,Y 410.703,Z 662.484,A -85,B 0,C 180,E1 10164.745,E2 10164.745} C_VEL
LIN {X 0,Y 412.257,Z 633.981,A -85,B 0,C 180,E1 10166.217,E2 10166.217} C_VEL
LIN {X 0,Y 413.053,Z 592.543,A -85,B 0,C 180,E1 10167.145,E2 10167.145} C_VEL
LIN {X 0,Y 412.774,Z 565.301,A -85,B 0,C 180,E1 10167.666,E2 10167.666} C_VEL
LIN {X 0,Y 402.236,Z 529.66,A -85,B 0,C 180,E1 10169.032,E2 10169.032} C_VEL
LIN {X 0,Y 402.159,Z 529.66,A -85,B 0,C 180,E1 10174.303,E2 10174.303} C_VEL
LIN {X 0,Y 401.802,Z 529.66,A -85,B 0,C 180,E1 10180.822,E2 10180.822} C_VEL
LIN {X 0,Y 401.561,Z 529.66,A -85,B 0,C 180,E1 10187.494,E2 10187.494} C_VEL
LIN {X 0,Y 401.28,Z 529.66,A -85,B 0,C 180,E1 10194.433,E2 10194.433} C_VEL
LIN {X 0,Y 401.096,Z 529.66,A -85,B 0,C 180,E1 10201.782,E2 10201.782} C_VEL
LIN {X 0,Y 401.035,Z 529.66,A -85,B 0,C 180,E1 10207.794,E2 10207.794} C_VEL
LIN {X 0,Y 401,Z 529.66,A -85,B 0,C 180,E1 10214.355,E2 10214.355} C_VEL
LIN {X 0,Y 400.997,Z 529.66,A -85,B 0,C 180,E1 10220.225,E2 10220.225} C_VEL
LIN {X 0,Y 401.083,Z 529.66,A -85,B 0,C 180,E1 10227.032,E2 10227.032} C_VEL
LIN {X 0,Y 419.412,Z 577.14,A -85,B 0,C 180,E1 10229.752,E2 10229.752} C_VEL
LIN {X 0,Y 420.143,Z 585.259,A -85,B 0,C 180,E1 10230.145,E2 10230.145} C_VEL
LIN {X 0,Y 417.11,Z 619.765,A -85,B 0,C 180,E1 10231.943,E2 10231.943} C_VEL
LIN {X 0,Y 413.385,Z 652.618,A -85,B 0,C 180,E1 10234.599,E2 10234.599} C_VEL
LIN {X 0,Y 409.65,Z 681.234,A -85,B 0,C 180,E1 10237.927,E2 10237.927} C_VEL
LIN {X 0,Y 406.584,Z 704.851,A -85,B 0,C 180,E1 10241.77,E2 10241.77} C_VEL
LIN {X 0,Y 404.441,Z 723.038,A -85,B 0,C 180,E1 10245.944,E2 10245.944} C_VEL
LIN {X 0,Y 403.285,Z 736.058,A -85,B 0,C 180,E1 10250.304,E2 10250.304} C_VEL
LIN {X 0,Y 402.777,Z 743.898,A -85,B 0,C 180,E1 10254.623,E2 10254.623} C_VEL
LIN {X 0,Y 402.563,Z 746.805,A -85,B 0,C 180,E1 10257.849,E2 10257.849} C_VEL
LIN {X 0,Y 402.712,Z 746.928,A -85,B 0,C 180,E1 10262.145,E2 10262.145} C_VEL
LIN {X 0,Y 402.87,Z 742.738,A -85,B 0,C 180,E1 10266.449,E2 10266.449} C_VEL
LIN {X 0,Y 403.727,Z 732.449,A -85,B 0,C 180,E1 10271.313,E2 10271.313} C_VEL
LIN {X 0,Y 405.517,Z 716.491,A -85,B 0,C 180,E1 10275.925,E2 10275.925} C_VEL
LIN {X 0,Y 408.099,Z 695.804,A -85,B 0,C 180,E1 10279.997,E2 10279.997} C_VEL
LIN {X 0,Y 411.568,Z 669.789,A -85,B 0,C 180,E1 10283.649,E2 10283.649} C_VEL
LIN {X 0,Y 415.554,Z 638.882,A -85,B 0,C 180,E1 10286.712,E2 10286.712} C_VEL
LIN {X 0,Y 419.3,Z 604.071,A -85,B 0,C 180,E1 10289.064,E2 10289.064} C_VEL
LIN {X 0,Y 420.743,Z 579.224,A -85,B 0,C 180,E1 10290.262,E2 10290.262} C_VEL
LIN {X 0,Y 412.271,Z 552.894,A -85,B 0,C 180,E1 10292.188,E2 10292.188} C_VEL
LIN {X 0,Y 402.966,Z 534.771,A -85,B 0,C 180,E1 10294.17,E2 10294.17} C_VEL
LIN {X 0,Y 401.059,Z 529.66,A -85,B 0,C 180,E1 10294.742,E2 10294.742} C_VEL
LIN {X 0,Y 400.887,Z 529.66,A -85,B 0,C 180,E1 10301.166,E2 10301.166} C_VEL
LIN {X 0,Y 400.968,Z 529.66,A -85,B 0,C 180,E1 10307.36,E2 10307.36} C_VEL
LIN {X 0,Y 401.058,Z 529.826,A -85,B 0,C 180,E1 10310.769,E2 10310.769} C_VEL
LIN {X 0,Y 403.604,Z 535.419,A -85,B 0,C 180,E1 10311.407,E2 10311.407} C_VEL
LIN {X 0,Y 413.797,Z 556.104,A -85,B 0,C 180,E1 10313.442,E2 10313.442} C_VEL
LIN {X 0,Y 421.956,Z 582.893,A -85,B 0,C 180,E1 10315.11,E2 10315.11} C_VEL
LIN {X 0,Y 423.001,Z 590.947,A -85,B 0,C 180,E1 10315.513,E2 10315.513} C_VEL
LIN {X 0,Y 419.79,Z 630.065,A -85,B 0,C 180,E1 10317.275,E2 10317.275} C_VEL
LIN {X 0,Y 415.853,Z 666.414,A -85,B 0,C 180,E1 10319.811,E2 10319.811} C_VEL
LIN {X 0,Y 411.826,Z 699.078,A -85,B 0,C 180,E1 10323.037,E2 10323.037} C_VEL
LIN {X 0,Y 410.604,Z 708.482,A -85,B 0,C 180,E1 10324.19,E2 10324.19} C_VEL
LIN {X 0,Y 405.278,Z 721.003,A -85,B 0,C 180,E1 10325.745,E2 10325.745} C_VEL
LIN {X 0,Y 399.839,Z 732.639,A -85,B 0,C 180,E1 10327.442,E2 10327.442} C_VEL
LIN {X 0,Y 397.203,Z 754.459,A -85,B 0,C 180,E1 10331.879,E2 10331.879} C_VEL
LIN {X 0,Y 395.557,Z 771.587,A -85,B 0,C 180,E1 10336.769,E2 10336.769} C_VEL
LIN {X 0,Y 394.952,Z 781.996,A -85,B 0,C 180,E1 10341.21,E2 10341.21} C_VEL
LIN {X 0,Y 394.72,Z 788.083,A -85,B 0,C 180,E1 10345.616,E2 10345.616} C_VEL
LIN {X 0,Y 394.69,Z 790.206,A -85,B 0,C 180,E1 10350.001,E2 10350.001} C_VEL
LIN {X 0,Y 394.76,Z 787.365,A -85,B 0,C 180,E1 10355.367,E2 10355.367} C_VEL
LIN {X 0,Y 395.082,Z 779.218,A -85,B 0,C 180,E1 10360.454,E2 10360.454} C_VEL
LIN {X 0,Y 396.177,Z 765.623,A -85,B 0,C 180,E1 10365.464,E2 10365.464} C_VEL
LIN {X 0,Y 398.568,Z 745.365,A -85,B 0,C 180,E1 10370.501,E2 10370.501} C_VEL
LIN {X 0,Y 402.019,Z 720.858,A -85,B 0,C 180,E1 10374.84,E2 10374.84} C_VEL
LIN {X 0,Y 406.343,Z 690.903,A -85,B 0,C 180,E1 10378.716,E2 10378.716} C_VEL
LIN {X 0,Y 410.83,Z 657.79,A -85,B 0,C 180,E1 10381.771,E2 10381.771} C_VEL
LIN {X 0,Y 415.036,Z 621.06,A -85,B 0,C 180,E1 10384.11,E2 10384.11} C_VEL
LIN {X 0,Y 417.134,Z 588.364,A -85,B 0,C 180,E1 10385.487,E2 10385.487} C_VEL
LIN {X 0,Y 396.063,Z 537.581,A -85,B 0,C 180,E1 10388.519,E2 10388.519} C_VEL
LIN {X 0,Y 393.174,Z 529.66,A -85,B 0,C 180,E1 10389.048,E2 10389.048} C_VEL
LIN {X 0,Y 393.065,Z 529.66,A -85,B 0,C 180,E1 10396.293,E2 10396.293} C_VEL
LIN {X 0,Y 393.13,Z 529.66,A -85,B 0,C 180,E1 10402.115,E2 10402.115} C_VEL
LIN {X 0,Y 393.203,Z 529.66,A -85,B 0,C 180,E1 10410.077,E2 10410.077} C_VEL
LIN {X 0,Y 393.463,Z 529.66,A -85,B 0,C 180,E1 10417.452,E2 10417.452} C_VEL
LIN {X 0,Y 393.659,Z 529.66,A -85,B 0,C 180,E1 10424.439,E2 10424.439} C_VEL
LIN {X 0,Y 393.96,Z 529.66,A -85,B 0,C 180,E1 10431.19,E2 10431.19} C_VEL
LIN {X 0,Y 394.474,Z 529.66,A -85,B 0,C 180,E1 10437.811,E2 10437.811} C_VEL
LIN {X 0,Y 394.266,Z 529.66,A -85,B 0,C 180,E1 10444.393,E2 10444.393} C_VEL
LIN {X 0,Y 393.934,Z 529.66,A -85,B 0,C 180,E1 10451.045,E2 10451.045} C_VEL
LIN {X 0,Y 393.657,Z 529.66,A -85,B 0,C 180,E1 10457.861,E2 10457.861} C_VEL
LIN {X 0,Y 393.349,Z 529.66,A -85,B 0,C 180,E1 10464.963,E2 10464.963} C_VEL
LIN {X 0,Y 393.137,Z 529.66,A -85,B 0,C 180,E1 10472.508,E2 10472.508} C_VEL
LIN {X 0,Y 393.135,Z 530.011,A -85,B 0,C 180,E1 10480.14,E2 10480.14} C_VEL
LIN {X 0,Y 406.585,Z 570.099,A -85,B 0,C 180,E1 10481.828,E2 10481.828} C_VEL
LIN {X 0,Y 405.304,Z 633.007,A -85,B 0,C 180,E1 10483.123,E2 10483.123} C_VEL
LIN {X 0,Y 403.592,Z 662.416,A -85,B 0,C 180,E1 10484.627,E2 10484.627} C_VEL
LIN {X 0,Y 401.296,Z 688.489,A -85,B 0,C 180,E1 10486.89,E2 10486.89} C_VEL
LIN {X 0,Y 398.678,Z 711.449,A -85,B 0,C 180,E1 10489.949,E2 10489.949} C_VEL
LIN {X 0,Y 396.828,Z 728.502,A -85,B 0,C 180,E1 10493.353,E2 10493.353} C_VEL
LIN {X 0,Y 395.682,Z 740.535,A -85,B 0,C 180,E1 10497.039,E2 10497.039} C_VEL
LIN {X 0,Y 395.031,Z 746.808,A -85,B 0,C 180,E1 10500.224,E2 10500.224} C_VEL
LIN {X 0,Y 394.598,Z 749.406,A -85,B 0,C 180,E1 10502.683,E2 10502.683} C_VEL
LIN {X 0,Y 394.405,Z 749.644,A -85,B 0,C 180,E1 10506.676,E2 10506.676} C_VEL
LIN {X 0,Y 395.21,Z 744.197,A -85,B 0,C 180,E1 10511.061,E2 10511.061} C_VEL
LIN {X 0,Y 396.185,Z 733.328,A -85,B 0,C 180,E1 10515.103,E2 10515.103} C_VEL
LIN {X 0,Y 397.852,Z 717.242,A -85,B 0,C 180,E1 10518.79,E2 10518.79} C_VEL
LIN {X 0,Y 400.117,Z 695.958,A -85,B 0,C 180,E1 10522.005,E2 10522.005} C_VEL
LIN {X 0,Y 402.581,Z 670.557,A -85,B 0,C 180,E1 10524.541,E2 10524.541} C_VEL
LIN {X 0,Y 404.497,Z 642.192,A -85,B 0,C 180,E1 10526.285,E2 10526.285} C_VEL
LIN {X 0,Y 405.505,Z 612.918,A -85,B 0,C 180,E1 10527.186,E2 10527.186} C_VEL
LIN {X 0,Y 405.435,Z 566.554,A -85,B 0,C 180,E1 10528.068,E2 10528.068} C_VEL
LIN {X 0,Y 394.399,Z 529.66,A -85,B 0,C 180,E1 10529.588,E2 10529.588} C_VEL
LIN {X 0,Y 394.173,Z 529.66,A -85,B 0,C 180,E1 10535.509,E2 10535.509} C_VEL
LIN {X 0,Y 393.879,Z 529.66,A -85,B 0,C 180,E1 10541.043,E2 10541.043} C_VEL
LIN {X 0,Y 393.618,Z 529.66,A -85,B 0,C 180,E1 10547.859,E2 10547.859} C_VEL
LIN {X 0,Y 393.338,Z 529.66,A -85,B 0,C 180,E1 10554.96,E2 10554.96} C_VEL
LIN {X 0,Y 393.146,Z 529.66,A -85,B 0,C 180,E1 10562.503,E2 10562.503} C_VEL
LIN {X 0,Y 393.125,Z 529.66,A -85,B 0,C 180,E1 10569.849,E2 10569.849} C_VEL
LIN {X 0,Y 393.073,Z 529.66,A -85,B 0,C 180,E1 10576.835,E2 10576.835} C_VEL
LIN {X 0,Y 393.042,Z 529.66,A -85,B 0,C 180,E1 10583.729,E2 10583.729} C_VEL
LIN {X 0,Y 393.154,Z 529.66,A -85,B 0,C 180,E1 10586.408,E2 10586.408} C_VEL
LIN {X 0,Y 411.568,Z 577.026,A -85,B 0,C 180,E1 10589.192,E2 10589.192} C_VEL
LIN {X 0,Y 413.139,Z 584.886,A -85,B 0,C 180,E1 10589.64,E2 10589.64} C_VEL
LIN {X 0,Y 409.917,Z 620.038,A -85,B 0,C 180,E1 10591.495,E2 10591.495} C_VEL
LIN {X 0,Y 406.143,Z 652.075,A -85,B 0,C 180,E1 10594.112,E2 10594.112} C_VEL
LIN {X 0,Y 402.339,Z 679.976,A -85,B 0,C 180,E1 10597.354,E2 10597.354} C_VEL
LIN {X 0,Y 399.016,Z 704.401,A -85,B 0,C 180,E1 10601.325,E2 10601.325} C_VEL
LIN {X 0,Y 396.708,Z 723.168,A -85,B 0,C 180,E1 10605.664,E2 10605.664} C_VEL
LIN {X 0,Y 395.436,Z 736.317,A -85,B 0,C 180,E1 10610.109,E2 10610.109} C_VEL
LIN {X 0,Y 394.921,Z 744.256,A -85,B 0,C 180,E1 10614.516,E2 10614.516} C_VEL
LIN {X 0,Y 394.673,Z 747.21,A -85,B 0,C 180,E1 10617.806,E2 10617.806} C_VEL
LIN {X 0,Y 394.822,Z 747.378,A -85,B 0,C 180,E1 10622.187,E2 10622.187} C_VEL
LIN {X 0,Y 395.02,Z 743.054,A -85,B 0,C 180,E1 10626.689,E2 10626.689} C_VEL
LIN {X 0,Y 395.945,Z 732.93,A -85,B 0,C 180,E1 10631.539,E2 10631.539} C_VEL
LIN {X 0,Y 397.871,Z 716.975,A -85,B 0,C 180,E1 10636.24,E2 10636.24} C_VEL
LIN {X 0,Y 400.637,Z 696.313,A -85,B 0,C 180,E1 10640.386,E2 10640.386} C_VEL
LIN {X 0,Y 404.328,Z 670.388,A -85,B 0,C 180,E1 10644.099,E2 10644.099} C_VEL
LIN {X 0,Y 408.553,Z 639.574,A -85,B 0,C 180,E1 10647.22,E2 10647.22} C_VEL
LIN {X 0,Y 412.661,Z 604.297,A -85,B 0,C 180,E1 10649.655,E2 10649.655} C_VEL
LIN {X 0,Y 414.143,Z 581.527,A -85,B 0,C 180,E1 10650.801,E2 10650.801} C_VEL
LIN {X 0,Y 406.523,Z 556.632,A -85,B 0,C 180,E1 10652.757,E2 10652.757} C_VEL
LIN {X 0,Y 397.995,Z 539.797,A -85,B 0,C 180,E1 10654.74,E2 10654.74} C_VEL
LIN {X 0,Y 394.362,Z 533.877,A -85,B 0,C 180,E1 10655.726,E2 10655.726} C_VEL
LIN {X 0,Y 393.107,Z 529.66,A -85,B 0,C 180,E1 10656.284,E2 10656.284} C_VEL
LIN {X 0,Y 393.002,Z 529.66,A -85,B 0,C 180,E1 10663.154,E2 10663.154} C_VEL
LIN {X 0,Y 393.059,Z 529.89,A -85,B 0,C 180,E1 10669.26,E2 10669.26} C_VEL
LIN {X 0,Y 395.637,Z 535.477,A -85,B 0,C 180,E1 10670.07,E2 10670.07} C_VEL
LIN {X 0,Y 404.205,Z 551.005,A -85,B 0,C 180,E1 10672.075,E2 10672.075} C_VEL
LIN {X 0,Y 412.766,Z 573.751,A -85,B 0,C 180,E1 10673.873,E2 10673.873} C_VEL
LIN {X 0,Y 416.377,Z 591.546,A -85,B 0,C 180,E1 10674.931,E2 10674.931} C_VEL
LIN {X 0,Y 412.89,Z 630.613,A -85,B 0,C 180,E1 10676.757,E2 10676.757} C_VEL
LIN {X 0,Y 408.649,Z 667.203,A -85,B 0,C 180,E1 10679.384,E2 10679.384} C_VEL
LIN {X 0,Y 404.238,Z 700.484,A -85,B 0,C 180,E1 10682.789,E2 10682.789} C_VEL
LIN {X 0,Y 400.421,Z 728.187,A -85,B 0,C 180,E1 10686.692,E2 10686.692} C_VEL
LIN {X 0,Y 399.839,Z 732.639,A -85,B 0,C 180,E1 10687.442,E2 10687.442} C_VEL
LIN {X 0,Y 394.485,Z 743.377,A -85,B 0,C 180,E1 10689.299,E2 10689.299} C_VEL
LIN {X 0,Y 389.56,Z 753.037,A -85,B 0,C 180,E1 10691.307,E2 10691.307} C_VEL
LIN {X 0,Y 387.88,Z 769.403,A -85,B 0,C 180,E1 10695.929,E2 10695.929} C_VEL
LIN {X 0,Y 387.064,Z 781.523,A -85,B 0,C 180,E1 10701.03,E2 10701.03} C_VEL
LIN {X 0,Y 386.852,Z 787.644,A -85,B 0,C 180,E1 10705.527,E2 10705.527} C_VEL
LIN {X 0,Y 386.826,Z 789.772,A -85,B 0,C 180,E1 10710.001,E2 10710.001} C_VEL
LIN {X 0,Y 386.875,Z 787.106,A -85,B 0,C 180,E1 10715.288,E2 10715.288} C_VEL
LIN {X 0,Y 387.161,Z 779.872,A -85,B 0,C 180,E1 10720.102,E2 10720.102} C_VEL
LIN {X 0,Y 388.176,Z 766.769,A -85,B 0,C 180,E1 10725.213,E2 10725.213} C_VEL
LIN {X 0,Y 390.258,Z 749,A -85,B 0,C 180,E1 10729.933,E2 10729.933} C_VEL
LIN {X 0,Y 393.553,Z 726.077,A -85,B 0,C 180,E1 10734.343,E2 10734.343} C_VEL
LIN {X 0,Y 397.873,Z 697.871,A -85,B 0,C 180,E1 10738.301,E2 10738.301} C_VEL
LIN {X 0,Y 402.491,Z 666.342,A -85,B 0,C 180,E1 10741.518,E2 10741.518} C_VEL
LIN {X 0,Y 407.013,Z 630.377,A -85,B 0,C 180,E1 10744.087,E2 10744.087} C_VEL
LIN {X 0,Y 410.515,Z 593.434,A -85,B 0,C 180,E1 10745.775,E2 10745.775} C_VEL
LIN {X 0,Y 400.001,Z 564.726,A -85,B 0,C 180,E1 10747.517,E2 10747.517} C_VEL
LIN {X 0,Y 385.231,Z 529.66,A -85,B 0,C 180,E1 10749.69,E2 10749.69} C_VEL
LIN {X 0,Y 385.065,Z 529.66,A -85,B 0,C 180,E1 10755.145,E2 10755.145} C_VEL
LIN {X 0,Y 385.189,Z 529.66,A -85,B 0,C 180,E1 10761.584,E2 10761.584} C_VEL
LIN {X 0,Y 385.14,Z 529.66,A -85,B 0,C 180,E1 10766.738,E2 10766.738} C_VEL
LIN {X 0,Y 385.365,Z 529.66,A -85,B 0,C 180,E1 10774.242,E2 10774.242} C_VEL
LIN {X 0,Y 385.664,Z 529.66,A -85,B 0,C 180,E1 10779.896,E2 10779.896} C_VEL
LIN {X 0,Y 385.821,Z 529.66,A -85,B 0,C 180,E1 10786.431,E2 10786.431} C_VEL
LIN {X 0,Y 386.231,Z 529.66,A -85,B 0,C 180,E1 10793.272,E2 10793.272} C_VEL
LIN {X 0,Y 386.53,Z 529.66,A -85,B 0,C 180,E1 10800.003,E2 10800.003} C_VEL
LIN {X 0,Y 386.227,Z 529.66,A -85,B 0,C 180,E1 10806.734,E2 10806.734} C_VEL
LIN {X 0,Y 385.938,Z 529.66,A -85,B 0,C 180,E1 10813.571,E2 10813.571} C_VEL
LIN {X 0,Y 385.603,Z 529.66,A -85,B 0,C 180,E1 10820.625,E2 10820.625} C_VEL
LIN {X 0,Y 385.28,Z 529.66,A -85,B 0,C 180,E1 10828.037,E2 10828.037} C_VEL
LIN {X 0,Y 385.092,Z 529.66,A -85,B 0,C 180,E1 10836.003,E2 10836.003} C_VEL
LIN {X 0,Y 385.176,Z 529.66,A -85,B 0,C 180,E1 10839.54,E2 10839.54} C_VEL
LIN {X 0,Y 399.352,Z 572.233,A -85,B 0,C 180,E1 10841.407,E2 10841.407} C_VEL
LIN {X 0,Y 398.032,Z 633.355,A -85,B 0,C 180,E1 10842.693,E2 10842.693} C_VEL
LIN {X 0,Y 396.248,Z 661.701,A -85,B 0,C 180,E1 10844.145,E2 10844.145} C_VEL
LIN {X 0,Y 393.94,Z 687.821,A -85,B 0,C 180,E1 10846.409,E2 10846.409} C_VEL
LIN {X 0,Y 391.359,Z 709.605,A -85,B 0,C 180,E1 10849.273,E2 10849.273} C_VEL
LIN {X 0,Y 389.232,Z 727.507,A -85,B 0,C 180,E1 10852.775,E2 10852.775} C_VEL
LIN {X 0,Y 387.972,Z 739.421,A -85,B 0,C 180,E1 10856.298,E2 10856.298} C_VEL
LIN {X 0,Y 387.269,Z 746.366,A -85,B 0,C 180,E1 10859.565,E2 10859.565} C_VEL
LIN {X 0,Y 386.519,Z 750.413,A -85,B 0,C 180,E1 10863.893,E2 10863.893} C_VEL
LIN {X 0,Y 386.733,Z 748.834,A -85,B 0,C 180,E1 10868.243,E2 10868.243} C_VEL
LIN {X 0,Y 387.595,Z 742.217,A -85,B 0,C 180,E1 10872.292,E2 10872.292} C_VEL
LIN {X 0,Y 388.748,Z 731.044,A -85,B 0,C 180,E1 10876.038,E2 10876.038} C_VEL
LIN {X 0,Y 390.658,Z 713.219,A -85,B 0,C 180,E1 10879.848,E2 10879.848} C_VEL
LIN {X 0,Y 393.203,Z 690.91,A -85,B 0,C 180,E1 10882.973,E2 10882.973} C_VEL
LIN {X 0,Y 395.672,Z 665.025,A -85,B 0,C 180,E1 10885.357,E2 10885.357} C_VEL
LIN {X 0,Y 397.423,Z 636.59,A -85,B 0,C 180,E1 10886.938,E2 10886.938} C_VEL
LIN {X 0,Y 398.364,Z 598.33,A -85,B 0,C 180,E1 10887.875,E2 10887.875} C_VEL
LIN {X 0,Y 398.145,Z 567.962,A -85,B 0,C 180,E1 10888.476,E2 10888.476} C_VEL
LIN {X 0,Y 386.534,Z 529.66,A -85,B 0,C 180,E1 10889.999,E2 10889.999} C_VEL
LIN {X 0,Y 386.264,Z 529.66,A -85,B 0,C 180,E1 10896.729,E2 10896.729} C_VEL
LIN {X 0,Y 385.851,Z 529.66,A -85,B 0,C 180,E1 10903.57,E2 10903.57} C_VEL
LIN {X 0,Y 385.583,Z 529.66,A -85,B 0,C 180,E1 10910.622,E2 10910.622} C_VEL
LIN {X 0,Y 385.264,Z 529.66,A -85,B 0,C 180,E1 10918.034,E2 10918.034} C_VEL
LIN {X 0,Y 385.175,Z 529.66,A -85,B 0,C 180,E1 10925.989,E2 10925.989} C_VEL
LIN {X 0,Y 385.093,Z 529.66,A -85,B 0,C 180,E1 10931.879,E2 10931.879} C_VEL
LIN {X 0,Y 385.085,Z 529.66,A -85,B 0,C 180,E1 10938.225,E2 10938.225} C_VEL
LIN {X 0,Y 385.171,Z 529.66,A -85,B 0,C 180,E1 10945.356,E2 10945.356} C_VEL
LIN {X 0,Y 385.283,Z 530.494,A -85,B 0,C 180,E1 10945.774,E2 10945.774} C_VEL
LIN {X 0,Y 403.884,Z 577.4,A -85,B 0,C 180,E1 10948.649,E2 10948.649} C_VEL
LIN {X 0,Y 405.954,Z 586.363,A -85,B 0,C 180,E1 10949.197,E2 10949.197} C_VEL
LIN {X 0,Y 402.536,Z 621.735,A -85,B 0,C 180,E1 10951.135,E2 10951.135} C_VEL
LIN {X 0,Y 398.539,Z 654.271,A -85,B 0,C 180,E1 10953.883,E2 10953.883} C_VEL
LIN {X 0,Y 394.489,Z 682.745,A -85,B 0,C 180,E1 10957.344,E2 10957.344} C_VEL
LIN {X 0,Y 391.158,Z 706.213,A -85,B 0,C 180,E1 10961.335,E2 10961.335} C_VEL
LIN {X 0,Y 388.788,Z 724.963,A -85,B 0,C 180,E1 10965.849,E2 10965.849} C_VEL
LIN {X 0,Y 387.508,Z 737.794,A -85,B 0,C 180,E1 10970.471,E2 10970.471} C_VEL
LIN {X 0,Y 386.937,Z 745.895,A -85,B 0,C 180,E1 10975.524,E2 10975.524} C_VEL
LIN {X 0,Y 386.851,Z 748.315,A -85,B 0,C 180,E1 10979.997,E2 10979.997} C_VEL
LIN {X 0,Y 386.977,Z 746.353,A -85,B 0,C 180,E1 10984.47,E2 10984.47} C_VEL
LIN {X 0,Y 387.597,Z 738.776,A -85,B 0,C 180,E1 10989.521,E2 10989.521} C_VEL
LIN {X 0,Y 389.089,Z 725.774,A -85,B 0,C 180,E1 10994.334,E2 10994.334} C_VEL
LIN {X 0,Y 391.596,Z 707.845,A -85,B 0,C 180,E1 10998.73,E2 10998.73} C_VEL
LIN {X 0,Y 395.243,Z 683.829,A -85,B 0,C 180,E1 11002.858,E2 11002.858} C_VEL
LIN {X 0,Y 399.565,Z 655.289,A -85,B 0,C 180,E1 11006.34,E2 11006.34} C_VEL
LIN {X 0,Y 403.832,Z 623.719,A -85,B 0,C 180,E1 11009.059,E2 11009.059} C_VEL
LIN {X 0,Y 407.965,Z 586.771,A -85,B 0,C 180,E1 11011.183,E2 11011.183} C_VEL
LIN {X 0,Y 402.027,Z 563.264,A -85,B 0,C 180,E1 11013.069,E2 11013.069} C_VEL
LIN {X 0,Y 393.603,Z 545.382,A -85,B 0,C 180,E1 11015.233,E2 11015.233} C_VEL
LIN {X 0,Y 387.957,Z 535.666,A -85,B 0,C 180,E1 11017.04,E2 11017.04} C_VEL
LIN {X 0,Y 385.159,Z 529.94,A -85,B 0,C 180,E1 11018.308,E2 11018.308} C_VEL
LIN {X 0,Y 385.024,Z 529.66,A -85,B 0,C 180,E1 11025.135,E2 11025.135} C_VEL
LIN {X 0,Y 385.163,Z 529.956,A -85,B 0,C 180,E1 11027.207,E2 11027.207} C_VEL
LIN {X 0,Y 387.689,Z 535.436,A -85,B 0,C 180,E1 11028.345,E2 11028.345} C_VEL
LIN {X 0,Y 390.161,Z 539.467,A -85,B 0,C 180,E1 11029.175,E2 11029.175} C_VEL
LIN {X 0,Y 397.557,Z 552.313,A -85,B 0,C 180,E1 11031.149,E2 11031.149} C_VEL
LIN {X 0,Y 405.822,Z 573.509,A -85,B 0,C 180,E1 11033.073,E2 11033.073} C_VEL
LIN {X 0,Y 409.758,Z 593.868,A -85,B 0,C 180,E1 11034.376,E2 11034.376} C_VEL
LIN {X 0,Y 405.717,Z 633.891,A -85,B 0,C 180,E1 11036.373,E2 11036.373} C_VEL
LIN {X 0,Y 401.12,Z 670.6,A -85,B 0,C 180,E1 11039.158,E2 11039.158} C_VEL
LIN {X 0,Y 396.671,Z 702.014,A -85,B 0,C 180,E1 11042.533,E2 11042.533} C_VEL
LIN {X 0,Y 392.696,Z 729.228,A -85,B 0,C 180,E1 11046.506,E2 11046.506} C_VEL
LIN {X 0,Y 389.724,Z 751.411,A -85,B 0,C 180,E1 11050.911,E2 11050.911} C_VEL
LIN {X 0,Y 389.56,Z 753.037,A -85,B 0,C 180,E1 11051.307,E2 11051.307} C_VEL
LIN {X 0,Y 387.874,Z 757.547,A -85,B 0,C 180,E1 11052.39,E2 11052.39} C_VEL
LIN {X 0,Y 380.186,Z 768.304,A -85,B 0,C 180,E1 11055.425,E2 11055.425} C_VEL
LIN {X 0,Y 380.011,Z 769.171,A -85,B 0,C 180,E1 11055.727,E2 11055.727} C_VEL
LIN {X 0,Y 379.182,Z 781.066,A -85,B 0,C 180,E1 11060.841,E2 11060.841} C_VEL
LIN {X 0,Y 378.962,Z 787.208,A -85,B 0,C 180,E1 11065.433,E2 11065.433} C_VEL
LIN {X 0,Y 378.936,Z 789.331,A -85,B 0,C 180,E1 11070.001,E2 11070.001} C_VEL
LIN {X 0,Y 378.966,Z 786.515,A -85,B 0,C 180,E1 11075.497,E2 11075.497} C_VEL
LIN {X 0,Y 379.337,Z 778.105,A -85,B 0,C 180,E1 11080.893,E2 11080.893} C_VEL
LIN {X 0,Y 380.628,Z 764.263,A -85,B 0,C 180,E1 11086.113,E2 11086.113} C_VEL
LIN {X 0,Y 383.288,Z 743.884,A -85,B 0,C 180,E1 11091.28,E2 11091.28} C_VEL
LIN {X 0,Y 386.994,Z 719.559,A -85,B 0,C 180,E1 11095.7,E2 11095.7} C_VEL
LIN {X 0,Y 391.63,Z 690.284,A -85,B 0,C 180,E1 11099.584,E2 11099.584} C_VEL
LIN {X 0,Y 396.37,Z 657.671,A -85,B 0,C 180,E1 11102.694,E2 11102.694} C_VEL
LIN {X 0,Y 400.871,Z 621.368,A -85,B 0,C 180,E1 11105.092,E2 11105.092} C_VEL
LIN {X 0,Y 402.92,Z 592.21,A -85,B 0,C 180,E1 11106.399,E2 11106.399} C_VEL
LIN {X 0,Y 384.32,Z 546.675,A -85,B 0,C 180,E1 11109.299,E2 11109.299} C_VEL
LIN {X 0,Y 377.3,Z 529.66,A -85,B 0,C 180,E1 11110.433,E2 11110.433} C_VEL
LIN {X 0,Y 377.079,Z 529.66,A -85,B 0,C 180,E1 11117.137,E2 11117.137} C_VEL
LIN {X 0,Y 377.202,Z 529.66,A -85,B 0,C 180,E1 11123.141,E2 11123.141} C_VEL
LIN {X 0,Y 377.229,Z 529.66,A -85,B 0,C 180,E1 11128.67,E2 11128.67} C_VEL
LIN {X 0,Y 377.425,Z 529.66,A -85,B 0,C 180,E1 11133.913,E2 11133.913} C_VEL
LIN {X 0,Y 377.638,Z 529.66,A -85,B 0,C 180,E1 11138.926,E2 11138.926} C_VEL
LIN {X 0,Y 377.875,Z 529.66,A -85,B 0,C 180,E1 11146.14,E2 11146.14} C_VEL
LIN {X 0,Y 378.309,Z 529.66,A -85,B 0,C 180,E1 11153.13,E2 11153.13} C_VEL
LIN {X 0,Y 378.628,Z 529.66,A -85,B 0,C 180,E1 11160.003,E2 11160.003} C_VEL
LIN {X 0,Y 378.309,Z 529.66,A -85,B 0,C 180,E1 11166.876,E2 11166.876} C_VEL
LIN {X 0,Y 377.99,Z 529.66,A -85,B 0,C 180,E1 11173.862,E2 11173.862} C_VEL
LIN {X 0,Y 377.632,Z 529.66,A -85,B 0,C 180,E1 11181.081,E2 11181.081} C_VEL
LIN {X 0,Y 377.321,Z 529.66,A -85,B 0,C 180,E1 11188.682,E2 11188.682} C_VEL
LIN {X 0,Y 377.159,Z 529.66,A -85,B 0,C 180,E1 11194.068,E2 11194.068} C_VEL
LIN {X 0,Y 377.26,Z 530.368,A -85,B 0,C 180,E1 11198.965,E2 11198.965} C_VEL
LIN {X 0,Y 392.163,Z 573.244,A -85,B 0,C 180,E1 11200.949,E2 11200.949} C_VEL
LIN {X 0,Y 390.829,Z 632.854,A -85,B 0,C 180,E1 11202.211,E2 11202.211} C_VEL
LIN {X 0,Y 388.897,Z 662.234,A -85,B 0,C 180,E1 11203.732,E2 11203.732} C_VEL
LIN {X 0,Y 386.428,Z 688.571,A -85,B 0,C 180,E1 11206.066,E2 11206.066} C_VEL
LIN {X 0,Y 383.597,Z 711.422,A -85,B 0,C 180,E1 11209.184,E2 11209.184} C_VEL
LIN {X 0,Y 381.316,Z 729.53,A -85,B 0,C 180,E1 11212.914,E2 11212.914} C_VEL
LIN {X 0,Y 379.988,Z 741.903,A -85,B 0,C 180,E1 11216.944,E2 11216.944} C_VEL
LIN {X 0,Y 378.994,Z 749.288,A -85,B 0,C 180,E1 11221.458,E2 11221.458} C_VEL
LIN {X 0,Y 378.618,Z 750.825,A -85,B 0,C 180,E1 11223.997,E2 11223.997} C_VEL
LIN {X 0,Y 378.765,Z 749.707,A -85,B 0,C 180,E1 11227.76,E2 11227.76} C_VEL
LIN {X 0,Y 379.662,Z 743.343,A -85,B 0,C 180,E1 11232.104,E2 11232.104} C_VEL
LIN {X 0,Y 380.953,Z 731.426,A -85,B 0,C 180,E1 11236.25,E2 11236.25} C_VEL
LIN {X 0,Y 382.972,Z 713.81,A -85,B 0,C 180,E1 11240.094,E2 11240.094} C_VEL
LIN {X 0,Y 385.582,Z 691.814,A -85,B 0,C 180,E1 11243.257,E2 11243.257} C_VEL
LIN {X 0,Y 388.156,Z 666.241,A -85,B 0,C 180,E1 11245.679,E2 11245.679} C_VEL
LIN {X 0,Y 390.055,Z 638.338,A -85,B 0,C 180,E1 11247.297,E2 11247.297} C_VEL
LIN {X 0,Y 390.971,Z 605.82,A -85,B 0,C 180,E1 11248.172,E2 11248.172} C_VEL
LIN {X 0,Y 390.997,Z 569.937,A -85,B 0,C 180,E1 11248.88,E2 11248.88} C_VEL
LIN {X 0,Y 378.6,Z 529.66,A -85,B 0,C 180,E1 11250.57,E2 11250.57} C_VEL
LIN {X 0,Y 378.339,Z 529.66,A -85,B 0,C 180,E1 11256.871,E2 11256.871} C_VEL
LIN {X 0,Y 377.905,Z 529.66,A -85,B 0,C 180,E1 11263.861,E2 11263.861} C_VEL
LIN {X 0,Y 377.613,Z 529.66,A -85,B 0,C 180,E1 11271.078,E2 11271.078} C_VEL
LIN {X 0,Y 377.309,Z 529.66,A -85,B 0,C 180,E1 11278.679,E2 11278.679} C_VEL
LIN {X 0,Y 377.209,Z 529.66,A -85,B 0,C 180,E1 11284.059,E2 11284.059} C_VEL
LIN {X 0,Y 377.126,Z 529.66,A -85,B 0,C 180,E1 11290.51,E2 11290.51} C_VEL
LIN {X 0,Y 377.082,Z 529.66,A -85,B 0,C 180,E1 11297.13,E2 11297.13} C_VEL
LIN {X 0,Y 377.225,Z 529.66,A -85,B 0,C 180,E1 11304.44,E2 11304.44} C_VEL
LIN {X 0,Y 377.297,Z 530.513,A -85,B 0,C 180,E1 11305.085,E2 11305.085} C_VEL
LIN {X 0,Y 396.401,Z 578.23,A -85,B 0,C 180,E1 11308.124,E2 11308.124} C_VEL
LIN {X 0,Y 398.732,Z 588.296,A -85,B 0,C 180,E1 11308.767,E2 11308.767} C_VEL
LIN {X 0,Y 395.111,Z 623.773,A -85,B 0,C 180,E1 11310.798,E2 11310.798} C_VEL
LIN {X 0,Y 390.934,Z 656.245,A -85,B 0,C 180,E1 11313.644,E2 11313.644} C_VEL
LIN {X 0,Y 386.899,Z 683.457,A -85,B 0,C 180,E1 11317.041,E2 11317.041} C_VEL
LIN {X 0,Y 383.414,Z 707.122,A -85,B 0,C 180,E1 11321.163,E2 11321.163} C_VEL
LIN {X 0,Y 380.963,Z 725.759,A -85,B 0,C 180,E1 11325.762,E2 11325.762} C_VEL
LIN {X 0,Y 379.593,Z 739.238,A -85,B 0,C 180,E1 11330.848,E2 11330.848} C_VEL
LIN {X 0,Y 379.055,Z 746.248,A -85,B 0,C 180,E1 11335.43,E2 11335.43} C_VEL
LIN {X 0,Y 378.962,Z 748.75,A -85,B 0,C 180,E1 11339.997,E2 11339.997} C_VEL
LIN {X 0,Y 379.104,Z 746.848,A -85,B 0,C 180,E1 11344.563,E2 11344.563} C_VEL
LIN {X 0,Y 379.777,Z 739.314,A -85,B 0,C 180,E1 11349.719,E2 11349.719} C_VEL
LIN {X 0,Y 381.508,Z 725.639,A -85,B 0,C 180,E1 11354.842,E2 11354.842} C_VEL
LIN {X 0,Y 384.267,Z 707.41,A -85,B 0,C 180,E1 11359.344,E2 11359.344} C_VEL
LIN {X 0,Y 388.279,Z 682.973,A -85,B 0,C 180,E1 11363.551,E2 11363.551} C_VEL
LIN {X 0,Y 392.783,Z 655.003,A -85,B 0,C 180,E1 11366.985,E2 11366.985} C_VEL
LIN {X 0,Y 397.501,Z 622.41,A -85,B 0,C 180,E1 11369.814,E2 11369.814} C_VEL
LIN {X 0,Y 401.28,Z 585.516,A -85,B 0,C 180,E1 11372.029,E2 11372.029} C_VEL
LIN {X 0,Y 395.034,Z 563.333,A -85,B 0,C 180,E1 11374.08,E2 11374.08} C_VEL
LIN {X 0,Y 387.224,Z 547.149,A -85,B 0,C 180,E1 11376.427,E2 11376.427} C_VEL
LIN {X 0,Y 383.278,Z 540.827,A -85,B 0,C 180,E1 11377.924,E2 11377.924} C_VEL
LIN {X 0,Y 381.189,Z 536.542,A -85,B 0,C 180,E1 11379.069,E2 11379.069} C_VEL
LIN {X 0,Y 377.889,Z 533.02,A -85,B 0,C 180,E1 11381.889,E2 11381.889} C_VEL
LIN {X 0,Y 378.687,Z 534.362,A -85,B 0,C 180,E1 11384.806,E2 11384.806} C_VEL
LIN {X 0,Y 382.098,Z 537.82,A -85,B 0,C 180,E1 11386.874,E2 11386.874} C_VEL
LIN {X 0,Y 388.556,Z 548.859,A -85,B 0,C 180,E1 11389.357,E2 11389.357} C_VEL
LIN {X 0,Y 396.484,Z 566.035,A -85,B 0,C 180,E1 11391.54,E2 11391.54} C_VEL
LIN {X 0,Y 402.563,Z 588.855,A -85,B 0,C 180,E1 11393.348,E2 11393.348} C_VEL
LIN {X 0,Y 403.205,Z 596.923,A -85,B 0,C 180,E1 11393.817,E2 11393.817} C_VEL
LIN {X 0,Y 398.722,Z 636.76,A -85,B 0,C 180,E1 11395.935,E2 11395.935} C_VEL
LIN {X 0,Y 393.779,Z 673.091,A -85,B 0,C 180,E1 11398.848,E2 11398.848} C_VEL
LIN {X 0,Y 388.913,Z 705.078,A -85,B 0,C 180,E1 11402.45,E2 11402.45} C_VEL
LIN {X 0,Y 384.749,Z 731.887,A -85,B 0,C 180,E1 11406.604,E2 11406.604} C_VEL
LIN {X 0,Y 381.7,Z 753.899,A -85,B 0,C 180,E1 11411.265,E2 11411.265} C_VEL
LIN {X 0,Y 380.011,Z 769.171,A -85,B 0,C 180,E1 11415.727,E2 11415.727} C_VEL
LIN {X 0,Y 378.494,Z 772.532,A -85,B 0,C 180,E1 11416.929,E2 11416.929} C_VEL
LIN {X 0,Y 371.446,Z 779.996,A -85,B 0,C 180,E1 11420.294,E2 11420.294} C_VEL
LIN {X 0,Y 371.313,Z 780.581,A -85,B 0,C 180,E1 11420.621,E2 11420.621} C_VEL
LIN {X 0,Y 371.072,Z 786.778,A -85,B 0,C 180,E1 11425.336,E2 11425.336} C_VEL
LIN {X 0,Y 371.046,Z 788.885,A -85,B 0,C 180,E1 11430.001,E2 11430.001} C_VEL
LIN {X 0,Y 371.062,Z 786.927,A -85,B 0,C 180,E1 11434.666,E2 11434.666} C_VEL
LIN {X 0,Y 371.37,Z 779.871,A -85,B 0,C 180,E1 11439.945,E2 11439.945} C_VEL
LIN {X 0,Y 372.422,Z 767.17,A -85,B 0,C 180,E1 11445.271,E2 11445.271} C_VEL
LIN {X 0,Y 374.699,Z 749.141,A -85,B 0,C 180,E1 11450.326,E2 11450.326} C_VEL
LIN {X 0,Y 378.381,Z 725.466,A -85,B 0,C 180,E1 11455.071,E2 11455.071} C_VEL
LIN {X 0,Y 383.116,Z 696.889,A -85,B 0,C 180,E1 11459.206,E2 11459.206} C_VEL
LIN {X 0,Y 388.047,Z 665.57,A -85,B 0,C 180,E1 11462.489,E2 11462.489} C_VEL
LIN {X 0,Y 392.85,Z 630.11,A -85,B 0,C 180,E1 11465.099,E2 11465.099} C_VEL
LIN {X 0,Y 395.918,Z 594.58,A -85,B 0,C 180,E1 11466.839,E2 11466.839} C_VEL
LIN {X 0,Y 379.1,Z 552.994,A -85,B 0,C 180,E1 11469.586,E2 11469.586} C_VEL
LIN {X 0,Y 369.275,Z 529.66,A -85,B 0,C 180,E1 11471.222,E2 11471.222} C_VEL
LIN {X 0,Y 369.16,Z 529.66,A -85,B 0,C 180,E1 11477.374,E2 11477.374} C_VEL
LIN {X 0,Y 369.197,Z 529.66,A -85,B 0,C 180,E1 11484.832,E2 11484.832} C_VEL
LIN {X 0,Y 369.335,Z 529.66,A -85,B 0,C 180,E1 11490.645,E2 11490.645} C_VEL
LIN {X 0,Y 369.554,Z 529.66,A -85,B 0,C 180,E1 11495.904,E2 11495.904} C_VEL
LIN {X 0,Y 369.857,Z 529.66,A -85,B 0,C 180,E1 11503.409,E2 11503.409} C_VEL
LIN {X 0,Y 370.154,Z 529.66,A -85,B 0,C 180,E1 11510.618,E2 11510.618} C_VEL
LIN {X 0,Y 370.747,Z 529.66,A -85,B 0,C 180,E1 11517.67,E2 11517.67} C_VEL
LIN {X 0,Y 370.54,Z 529.66,A -85,B 0,C 180,E1 11524.675,E2 11524.675} C_VEL
LIN {X 0,Y 370.152,Z 529.66,A -85,B 0,C 180,E1 11531.924,E2 11531.924} C_VEL
LIN {X 0,Y 369.787,Z 529.66,A -85,B 0,C 180,E1 11539.057,E2 11539.057} C_VEL
LIN {X 0,Y 369.442,Z 529.66,A -85,B 0,C 180,E1 11546.702,E2 11546.702} C_VEL
LIN {X 0,Y 369.246,Z 529.66,A -85,B 0,C 180,E1 11552.094,E2 11552.094} C_VEL
LIN {X 0,Y 369.36,Z 530.407,A -85,B 0,C 180,E1 11558.331,E2 11558.331} C_VEL
LIN {X 0,Y 384.992,Z 574.872,A -85,B 0,C 180,E1 11560.482,E2 11560.482} C_VEL
LIN {X 0,Y 383.614,Z 633.25,A -85,B 0,C 180,E1 11561.745,E2 11561.745} C_VEL
LIN {X 0,Y 381.6,Z 662.495,A -85,B 0,C 180,E1 11563.282,E2 11563.282} C_VEL
LIN {X 0,Y 378.983,Z 689.127,A -85,B 0,C 180,E1 11565.685,E2 11565.685} C_VEL
LIN {X 0,Y 376.175,Z 710.505,A -85,B 0,C 180,E1 11568.619,E2 11568.619} C_VEL
LIN {X 0,Y 373.719,Z 728.836,A -85,B 0,C 180,E1 11572.376,E2 11572.376} C_VEL
LIN {X 0,Y 372.273,Z 740.996,A -85,B 0,C 180,E1 11576.219,E2 11576.219} C_VEL
LIN {X 0,Y 371.483,Z 747.673,A -85,B 0,C 180,E1 11579.653,E2 11579.653} C_VEL
LIN {X 0,Y 370.747,Z 751.09,A -85,B 0,C 180,E1 11583.569,E2 11583.569} C_VEL
LIN {X 0,Y 370.691,Z 751.14,A -85,B 0,C 180,E1 11585.978,E2 11585.978} C_VEL
LIN {X 0,Y 371.355,Z 747.445,A -85,B 0,C 180,E1 11590.144,E2 11590.144} C_VEL
LIN {X 0,Y 372.319,Z 739.2,A -85,B 0,C 180,E1 11594.122,E2 11594.122} C_VEL
LIN {X 0,Y 373.932,Z 725.467,A -85,B 0,C 180,E1 11598.087,E2 11598.087} C_VEL
LIN {X 0,Y 376.296,Z 706.658,A -85,B 0,C 180,E1 11601.64,E2 11601.64} C_VEL
LIN {X 0,Y 379.119,Z 683.03,A -85,B 0,C 180,E1 11604.627,E2 11604.627} C_VEL
LIN {X 0,Y 381.499,Z 656.19,A -85,B 0,C 180,E1 11606.81,E2 11606.81} C_VEL
LIN {X 0,Y 383.243,Z 626.779,A -85,B 0,C 180,E1 11608.157,E2 11608.157} C_VEL
LIN {X 0,Y 383.513,Z 570.545,A -85,B 0,C 180,E1 11609.349,E2 11609.349} C_VEL
LIN {X 0,Y 370.725,Z 529.66,A -85,B 0,C 180,E1 11611.166,E2 11611.166} C_VEL
LIN {X 0,Y 370.403,Z 529.66,A -85,B 0,C 180,E1 11617.019,E2 11617.019} C_VEL
LIN {X 0,Y 369.974,Z 529.66,A -85,B 0,C 180,E1 11624.164,E2 11624.164} C_VEL
LIN {X 0,Y 369.676,Z 529.66,A -85,B 0,C 180,E1 11631.553,E2 11631.553} C_VEL
LIN {X 0,Y 369.437,Z 529.66,A -85,B 0,C 180,E1 11636.698,E2 11636.698} C_VEL
LIN {X 0,Y 369.262,Z 529.66,A -85,B 0,C 180,E1 11642.088,E2 11642.088} C_VEL
LIN {X 0,Y 369.168,Z 529.66,A -85,B 0,C 180,E1 11649.042,E2 11649.042} C_VEL
LIN {X 0,Y 369.177,Z 529.66,A -85,B 0,C 180,E1 11655.98,E2 11655.98} C_VEL
LIN {X 0,Y 369.268,Z 529.66,A -85,B 0,C 180,E1 11663.556,E2 11663.556} C_VEL
LIN {X 0,Y 369.348,Z 530.136,A -85,B 0,C 180,E1 11664.373,E2 11664.373} C_VEL
LIN {X 0,Y 388.794,Z 578.944,A -85,B 0,C 180,E1 11667.576,E2 11667.576} C_VEL
LIN {X 0,Y 391.564,Z 589.695,A -85,B 0,C 180,E1 11668.307,E2 11668.307} C_VEL
LIN {X 0,Y 387.767,Z 625.388,A -85,B 0,C 180,E1 11670.426,E2 11670.426} C_VEL
LIN {X 0,Y 383.341,Z 658.125,A -85,B 0,C 180,E1 11673.396,E2 11673.396} C_VEL
LIN {X 0,Y 379.197,Z 685.013,A -85,B 0,C 180,E1 11676.858,E2 11676.858} C_VEL
LIN {X 0,Y 375.644,Z 708.093,A -85,B 0,C 180,E1 11681.005,E2 11681.005} C_VEL
LIN {X 0,Y 373.232,Z 725.466,A -85,B 0,C 180,E1 11685.36,E2 11685.36} C_VEL
LIN {X 0,Y 371.843,Z 738.253,A -85,B 0,C 180,E1 11690.065,E2 11690.065} C_VEL
LIN {X 0,Y 371.188,Z 746.591,A -85,B 0,C 180,E1 11695.333,E2 11695.333} C_VEL
LIN {X 0,Y 371.073,Z 749.184,A -85,B 0,C 180,E1 11699.997,E2 11699.997} C_VEL
LIN {X 0,Y 371.261,Z 747.358,A -85,B 0,C 180,E1 11704.66,E2 11704.66} C_VEL
LIN {X 0,Y 371.978,Z 739.882,A -85,B 0,C 180,E1 11709.925,E2 11709.925} C_VEL
LIN {X 0,Y 373.722,Z 727.187,A -85,B 0,C 180,E1 11714.882,E2 11714.882} C_VEL
LIN {X 0,Y 376.807,Z 708.146,A -85,B 0,C 180,E1 11719.743,E2 11719.743} C_VEL
LIN {X 0,Y 381.113,Z 683.786,A -85,B 0,C 180,E1 11724.039,E2 11724.039} C_VEL
LIN {X 0,Y 386.097,Z 654.943,A -85,B 0,C 180,E1 11727.649,E2 11727.649} C_VEL
LIN {X 0,Y 391.244,Z 621.756,A -85,B 0,C 180,E1 11730.569,E2 11730.569} C_VEL
LIN {X 0,Y 395.099,Z 587.914,A -85,B 0,C 180,E1 11732.673,E2 11732.673} C_VEL
LIN {X 0,Y 389.941,Z 567.805,A -85,B 0,C 180,E1 11734.683,E2 11734.683} C_VEL
LIN {X 0,Y 383.021,Z 552.564,A -85,B 0,C 180,E1 11737.065,E2 11737.065} C_VEL
LIN {X 0,Y 378.208,Z 543.661,A -85,B 0,C 180,E1 11739.49,E2 11739.49} C_VEL
LIN {X 0,Y 375.616,Z 540.513,A -85,B 0,C 180,E1 11742.424,E2 11742.424} C_VEL
LIN {X 0,Y 377.546,Z 543.038,A -85,B 0,C 180,E1 11745.534,E2 11745.534} C_VEL
LIN {X 0,Y 379.42,Z 545.741,A -85,B 0,C 180,E1 11746.666,E2 11746.666} C_VEL
LIN {X 0,Y 385.012,Z 555.692,A -85,B 0,C 180,E1 11748.974,E2 11748.974} C_VEL
LIN {X 0,Y 391.733,Z 571.37,A -85,B 0,C 180,E1 11751.04,E2 11751.04} C_VEL
LIN {X 0,Y 397.098,Z 595.13,A -85,B 0,C 180,E1 11753.002,E2 11753.002} C_VEL
LIN {X 0,Y 392.337,Z 635.648,A -85,B 0,C 180,E1 11755.205,E2 11755.205} C_VEL
LIN {X 0,Y 386.857,Z 672.767,A -85,B 0,C 180,E1 11758.226,E2 11758.226} C_VEL
LIN {X 0,Y 381.754,Z 704.412,A -85,B 0,C 180,E1 11761.86,E2 11761.86} C_VEL
LIN {X 0,Y 377.293,Z 731.386,A -85,B 0,C 180,E1 11766.113,E2 11766.113} C_VEL
LIN {X 0,Y 373.997,Z 753.408,A -85,B 0,C 180,E1 11770.864,E2 11770.864} C_VEL
LIN {X 0,Y 372.076,Z 770.105,A -85,B 0,C 180,E1 11775.918,E2 11775.918} C_VEL
LIN {X 0,Y 371.313,Z 780.581,A -85,B 0,C 180,E1 11780.621,E2 11780.621} C_VEL
LIN {X 0,Y 368.671,Z 783.664,A -85,B 0,C 180,E1 11782.556,E2 11782.556} C_VEL
LIN {X 0,Y 363.113,Z 786.851,A -85,B 0,C 180,E1 11785.869,E2 11785.869} C_VEL
LIN {X 0,Y 363.157,Z 788.434,A -85,B 0,C 180,E1 11790.001,E2 11790.001} C_VEL
LIN {X 0,Y 363.175,Z 786.442,A -85,B 0,C 180,E1 11794.768,E2 11794.768} C_VEL
LIN {X 0,Y 363.51,Z 779.289,A -85,B 0,C 180,E1 11800.163,E2 11800.163} C_VEL
LIN {X 0,Y 364.646,Z 766.407,A -85,B 0,C 180,E1 11805.605,E2 11805.605} C_VEL
LIN {X 0,Y 367.112,Z 748.187,A -85,B 0,C 180,E1 11810.765,E2 11810.765} C_VEL
LIN {X 0,Y 370.973,Z 724.224,A -85,B 0,C 180,E1 11815.608,E2 11815.608} C_VEL
LIN {X 0,Y 375.669,Z 696.766,A -85,B 0,C 180,E1 11819.625,E2 11819.625} C_VEL
LIN {X 0,Y 380.848,Z 664.968,A -85,B 0,C 180,E1 11823.012,E2 11823.012} C_VEL
LIN {X 0,Y 385.846,Z 628.993,A -85,B 0,C 180,E1 11825.681,E2 11825.681} C_VEL
LIN {X 0,Y 388.629,Z 596.041,A -85,B 0,C 180,E1 11827.347,E2 11827.347} C_VEL
LIN {X 0,Y 372.054,Z 554.927,A -85,B 0,C 180,E1 11830.163,E2 11830.163} C_VEL
LIN {X 0,Y 361.306,Z 529.66,A -85,B 0,C 180,E1 11831.933,E2 11831.933} C_VEL
LIN {X 0,Y 361.252,Z 529.66,A -85,B 0,C 180,E1 11838.755,E2 11838.755} C_VEL
LIN {X 0,Y 361.221,Z 529.66,A -85,B 0,C 180,E1 11844.212,E2 11844.212} C_VEL
LIN {X 0,Y 361.396,Z 529.66,A -85,B 0,C 180,E1 11851.266,E2 11851.266} C_VEL
LIN {X 0,Y 361.709,Z 529.66,A -85,B 0,C 180,E1 11857.951,E2 11857.951} C_VEL
LIN {X 0,Y 361.996,Z 529.66,A -85,B 0,C 180,E1 11865.519,E2 11865.519} C_VEL
LIN {X 0,Y 362.454,Z 529.66,A -85,B 0,C 180,E1 11872.828,E2 11872.828} C_VEL
LIN {X 0,Y 362.849,Z 529.66,A -85,B 0,C 180,E1 11880.003,E2 11880.003} C_VEL
LIN {X 0,Y 362.463,Z 529.66,A -85,B 0,C 180,E1 11887.178,E2 11887.178} C_VEL
LIN {X 0,Y 362.095,Z 529.66,A -85,B 0,C 180,E1 11894.483,E2 11894.483} C_VEL
LIN {X 0,Y 361.703,Z 529.66,A -85,B 0,C 180,E1 11902.057,E2 11902.057} C_VEL
LIN {X 0,Y 361.36,Z 529.66,A -85,B 0,C 180,E1 11910.076,E2 11910.076} C_VEL
LIN {X 0,Y 361.342,Z 529.66,A -85,B 0,C 180,E1 11917.603,E2 11917.603} C_VEL
LIN {X 0,Y 377.676,Z 575.269,A -85,B 0,C 180,E1 11919.957,E2 11919.957} C_VEL
LIN {X 0,Y 376.359,Z 634.755,A -85,B 0,C 180,E1 11921.303,E2 11921.303} C_VEL
LIN {X 0,Y 374.24,Z 663.892,A -85,B 0,C 180,E1 11922.896,E2 11922.896} C_VEL
LIN {X 0,Y 371.451,Z 690.301,A -85,B 0,C 180,E1 11925.362,E2 11925.362} C_VEL
LIN {X 0,Y 368.361,Z 712.776,A -85,B 0,C 180,E1 11928.586,E2 11928.586} C_VEL
LIN {X 0,Y 365.807,Z 730.731,A -85,B 0,C 180,E1 11932.482,E2 11932.482} C_VEL
LIN {X 0,Y 364.32,Z 742.868,A -85,B 0,C 180,E1 11936.654,E2 11936.654} C_VEL
LIN {X 0,Y 363.404,Z 749.498,A -85,B 0,C 180,E1 11940.697,E2 11940.697} C_VEL
LIN {X 0,Y 362.767,Z 751.628,A -85,B 0,C 180,E1 11945.419,E2 11945.419} C_VEL
LIN {X 0,Y 363.399,Z 748.464,A -85,B 0,C 180,E1 11949.752,E2 11949.752} C_VEL
LIN {X 0,Y 364.529,Z 739.35,A -85,B 0,C 180,E1 11954.39,E2 11954.39} C_VEL
LIN {X 0,Y 366.36,Z 724.283,A -85,B 0,C 180,E1 11958.709,E2 11958.709} C_VEL
LIN {X 0,Y 369.009,Z 704.558,A -85,B 0,C 180,E1 11962.362,E2 11962.362} C_VEL
LIN {X 0,Y 372.009,Z 680.065,A -85,B 0,C 180,E1 11965.346,E2 11965.346} C_VEL
LIN {X 0,Y 374.494,Z 652.722,A -85,B 0,C 180,E1 11967.473,E2 11967.473} C_VEL
LIN {X 0,Y 376.056,Z 623.411,A -85,B 0,C 180,E1 11968.714,E2 11968.714} C_VEL
LIN {X 0,Y 376.428,Z 572.612,A -85,B 0,C 180,E1 11969.777,E2 11969.777} C_VEL
LIN {X 0,Y 362.83,Z 529.66,A -85,B 0,C 180,E1 11971.786,E2 11971.786} C_VEL
LIN {X 0,Y 362.257,Z 529.66,A -85,B 0,C 180,E1 11979.59,E2 11979.59} C_VEL
LIN {X 0,Y 361.909,Z 529.66,A -85,B 0,C 180,E1 11986.969,E2 11986.969} C_VEL
LIN {X 0,Y 361.591,Z 529.66,A -85,B 0,C 180,E1 11994.664,E2 11994.664} C_VEL
LIN {X 0,Y 361.358,Z 529.66,A -85,B 0,C 180,E1 12000.072,E2 12000.072} C_VEL
LIN {X 0,Y 361.245,Z 529.66,A -85,B 0,C 180,E1 12007.466,E2 12007.466} C_VEL
LIN {X 0,Y 361.256,Z 529.66,A -85,B 0,C 180,E1 12014.753,E2 12014.753} C_VEL
LIN {X 0,Y 361.23,Z 529.66,A -85,B 0,C 180,E1 12021.196,E2 12021.196} C_VEL
LIN {X 0,Y 361.396,Z 529.66,A -85,B 0,C 180,E1 12023.623,E2 12023.623} C_VEL
LIN {X 0,Y 381.158,Z 579.559,A -85,B 0,C 180,E1 12027.008,E2 12027.008} C_VEL
LIN {X 0,Y 384.385,Z 591.536,A -85,B 0,C 180,E1 12027.857,E2 12027.857} C_VEL
LIN {X 0,Y 380.423,Z 626.966,A -85,B 0,C 180,E1 12030.043,E2 12030.043} C_VEL
LIN {X 0,Y 375.923,Z 658.638,A -85,B 0,C 180,E1 12032.99,E2 12032.99} C_VEL
LIN {X 0,Y 371.482,Z 686.456,A -85,B 0,C 180,E1 12036.665,E2 12036.665} C_VEL
LIN {X 0,Y 367.654,Z 710.405,A -85,B 0,C 180,E1 12041.139,E2 12041.139} C_VEL
LIN {X 0,Y 365.263,Z 727.404,A -85,B 0,C 180,E1 12045.645,E2 12045.645} C_VEL
LIN {X 0,Y 363.905,Z 739.674,A -85,B 0,C 180,E1 12050.449,E2 12050.449} C_VEL
LIN {X 0,Y 363.294,Z 747.168,A -85,B 0,C 180,E1 12055.454,E2 12055.454} C_VEL
LIN {X 0,Y 363.184,Z 749.616,A -85,B 0,C 180,E1 12059.997,E2 12059.997} C_VEL
LIN {X 0,Y 363.405,Z 747.882,A -85,B 0,C 180,E1 12064.761,E2 12064.761} C_VEL
LIN {X 0,Y 364.18,Z 740.484,A -85,B 0,C 180,E1 12070.139,E2 12070.139} C_VEL
LIN {X 0,Y 365.934,Z 728.716,A -85,B 0,C 180,E1 12074.932,E2 12074.932} C_VEL
LIN {X 0,Y 369.17,Z 709.987,A -85,B 0,C 180,E1 12079.929,E2 12079.929} C_VEL
LIN {X 0,Y 373.698,Z 686.327,A -85,B 0,C 180,E1 12084.302,E2 12084.302} C_VEL
LIN {X 0,Y 379.028,Z 657.833,A -85,B 0,C 180,E1 12088.049,E2 12088.049} C_VEL
LIN {X 0,Y 384.58,Z 625.115,A -85,B 0,C 180,E1 12091.079,E2 12091.079} C_VEL
LIN {X 0,Y 389.129,Z 590.534,A -85,B 0,C 180,E1 12093.336,E2 12093.336} C_VEL
LIN {X 0,Y 384.431,Z 570.682,A -85,B 0,C 180,E1 12095.512,E2 12095.512} C_VEL
LIN {X 0,Y 378.349,Z 556.258,A -85,B 0,C 180,E1 12098.093,E2 12098.093} C_VEL
LIN {X 0,Y 375.259,Z 550.737,A -85,B 0,C 180,E1 12099.971,E2 12099.971} C_VEL
LIN {X 0,Y 373.517,Z 548.128,A -85,B 0,C 180,E1 12102.443,E2 12102.443} C_VEL
LIN {X 0,Y 375.43,Z 550.678,A -85,B 0,C 180,E1 12105.5,E2 12105.5} C_VEL
LIN {X 0,Y 379.43,Z 558.292,A -85,B 0,C 180,E1 12107.739,E2 12107.739} C_VEL
LIN {X 0,Y 385.405,Z 571.762,A -85,B 0,C 180,E1 12109.955,E2 12109.955} C_VEL
LIN {X 0,Y 390.144,Z 591.589,A -85,B 0,C 180,E1 12111.874,E2 12111.874} C_VEL
LIN {X 0,Y 390.578,Z 601.35,A -85,B 0,C 180,E1 12112.53,E2 12112.53} C_VEL
LIN {X 0,Y 385.176,Z 640.699,A -85,B 0,C 180,E1 12114.853,E2 12114.853} C_VEL
LIN {X 0,Y 379.41,Z 677.019,A -85,B 0,C 180,E1 12118.032,E2 12118.032} C_VEL
LIN {X 0,Y 373.803,Z 708.457,A -85,B 0,C 180,E1 12121.899,E2 12121.899} C_VEL
LIN {X 0,Y 369.151,Z 735.29,A -85,B 0,C 180,E1 12126.432,E2 12126.432} C_VEL
LIN {X 0,Y 365.775,Z 757.172,A -85,B 0,C 180,E1 12131.584,E2 12131.584} C_VEL
LIN {X 0,Y 364.026,Z 772.121,A -85,B 0,C 180,E1 12136.573,E2 12136.573} C_VEL
LIN {X 0,Y 363.331,Z 782.133,A -85,B 0,C 180,E1 12141.643,E2 12141.643} C_VEL
LIN {X 0,Y 363.113,Z 786.851,A -85,B 0,C 180,E1 12145.869,E2 12145.869} C_VEL
LIN {X 0,Y 360.507,Z 787.909,A -85,B 0,C 180,E1 12147.896,E2 12147.896} C_VEL
LIN {X 0,Y 355.211,Z 787.855,A -85,B 0,C 180,E1 12151.227,E2 12151.227} C_VEL
LIN {X 0,Y 355.206,Z 787.688,A -85,B 0,C 180,E1 12151.316,E2 12151.316} C_VEL
LIN {X 0,Y 355.269,Z 784.746,A -85,B 0,C 180,E1 12156.097,E2 12156.097} C_VEL
LIN {X 0,Y 355.788,Z 776.256,A -85,B 0,C 180,E1 12161.623,E2 12161.623} C_VEL
LIN {X 0,Y 357.271,Z 761.887,A -85,B 0,C 180,E1 12167.198,E2 12167.198} C_VEL
LIN {X 0,Y 360.102,Z 743.186,A -85,B 0,C 180,E1 12172.158,E2 12172.158} C_VEL
LIN {X 0,Y 364.262,Z 719.17,A -85,B 0,C 180,E1 12176.777,E2 12176.777} C_VEL
LIN {X 0,Y 369.615,Z 689.015,A -85,B 0,C 180,E1 12180.987,E2 12180.987} C_VEL
LIN {X 0,Y 375.022,Z 655.758,A -85,B 0,C 180,E1 12184.287,E2 12184.287} C_VEL
LIN {X 0,Y 379.969,Z 619.194,A -85,B 0,C 180,E1 12186.775,E2 12186.775} C_VEL
LIN {X 0,Y 381.492,Z 597.987,A -85,B 0,C 180,E1 12187.833,E2 12187.833} C_VEL
LIN {X 0,Y 365.179,Z 557.432,A -85,B 0,C 180,E1 12190.718,E2 12190.718} C_VEL
LIN {X 0,Y 353.305,Z 529.66,A -85,B 0,C 180,E1 12192.701,E2 12192.701} C_VEL
LIN {X 0,Y 353.289,Z 529.66,A -85,B 0,C 180,E1 12200.25,E2 12200.25} C_VEL
LIN {X 0,Y 353.33,Z 529.66,A -85,B 0,C 180,E1 12206.28,E2 12206.28} C_VEL
LIN {X 0,Y 353.533,Z 529.66,A -85,B 0,C 180,E1 12213.684,E2 12213.684} C_VEL
LIN {X 0,Y 353.852,Z 529.66,A -85,B 0,C 180,E1 12220.056,E2 12220.056} C_VEL
LIN {X 0,Y 354.214,Z 529.66,A -85,B 0,C 180,E1 12227.705,E2 12227.705} C_VEL
LIN {X 0,Y 354.678,Z 529.66,A -85,B 0,C 180,E1 12235.122,E2 12235.122} C_VEL
LIN {X 0,Y 354.953,Z 529.66,A -85,B 0,C 180,E1 12240.003,E2 12240.003} C_VEL
LIN {X 0,Y 354.529,Z 529.66,A -85,B 0,C 180,E1 12247.339,E2 12247.339} C_VEL
LIN {X 0,Y 354.169,Z 529.66,A -85,B 0,C 180,E1 12254.815,E2 12254.815} C_VEL
LIN {X 0,Y 353.755,Z 529.66,A -85,B 0,C 180,E1 12262.579,E2 12262.579} C_VEL
LIN {X 0,Y 353.479,Z 529.66,A -85,B 0,C 180,E1 12268.011,E2 12268.011} C_VEL
LIN {X 0,Y 353.296,Z 529.66,A -85,B 0,C 180,E1 12275.753,E2 12275.753} C_VEL
LIN {X 0,Y 353.411,Z 530.359,A -85,B 0,C 180,E1 12276.932,E2 12276.932} C_VEL
LIN {X 0,Y 370.451,Z 576.415,A -85,B 0,C 180,E1 12279.429,E2 12279.429} C_VEL
LIN {X 0,Y 369.25,Z 634.212,A -85,B 0,C 180,E1 12280.758,E2 12280.758} C_VEL
LIN {X 0,Y 367.189,Z 662.519,A -85,B 0,C 180,E1 12282.291,E2 12282.291} C_VEL
LIN {X 0,Y 364.23,Z 689.421,A -85,B 0,C 180,E1 12284.777,E2 12284.777} C_VEL
LIN {X 0,Y 360.959,Z 712.055,A -85,B 0,C 180,E1 12288.018,E2 12288.018} C_VEL
LIN {X 0,Y 358.283,Z 729.787,A -85,B 0,C 180,E1 12291.833,E2 12291.833} C_VEL
LIN {X 0,Y 356.64,Z 741.876,A -85,B 0,C 180,E1 12295.838,E2 12295.838} C_VEL
LIN {X 0,Y 355.752,Z 748.476,A -85,B 0,C 180,E1 12299.401,E2 12299.401} C_VEL
LIN {X 0,Y 354.996,Z 751.762,A -85,B 0,C 180,E1 12303.214,E2 12303.214} C_VEL
LIN {X 0,Y 355.031,Z 751.133,A -85,B 0,C 180,E1 12307.509,E2 12307.509} C_VEL
LIN {X 0,Y 355.995,Z 745.328,A -85,B 0,C 180,E1 12312.072,E2 12312.072} C_VEL
LIN {X 0,Y 357.508,Z 733.573,A -85,B 0,C 180,E1 12316.644,E2 12316.644} C_VEL
LIN {X 0,Y 359.733,Z 716.858,A -85,B 0,C 180,E1 12320.644,E2 12320.644} C_VEL
LIN {X 0,Y 362.767,Z 694.933,A -85,B 0,C 180,E1 12324.115,E2 12324.115} C_VEL
LIN {X 0,Y 365.743,Z 669.512,A -85,B 0,C 180,E1 12326.747,E2 12326.747} C_VEL
LIN {X 0,Y 367.977,Z 641.513,A -85,B 0,C 180,E1 12328.53,E2 12328.53} C_VEL
LIN {X 0,Y 369.114,Z 610.138,A -85,B 0,C 180,E1 12329.487,E2 12329.487} C_VEL
LIN {X 0,Y 369.333,Z 574.524,A -85,B 0,C 180,E1 12330.227,E2 12330.227} C_VEL
LIN {X 0,Y 354.957,Z 529.66,A -85,B 0,C 180,E1 12332.33,E2 12332.33} C_VEL
LIN {X 0,Y 354.321,Z 529.66,A -85,B 0,C 180,E1 12339.807,E2 12339.807} C_VEL
LIN {X 0,Y 353.947,Z 529.66,A -85,B 0,C 180,E1 12347.362,E2 12347.362} C_VEL
LIN {X 0,Y 353.586,Z 529.66,A -85,B 0,C 180,E1 12355.261,E2 12355.261} C_VEL
LIN {X 0,Y 353.334,Z 529.66,A -85,B 0,C 180,E1 12361.33,E2 12361.33} C_VEL
LIN {X 0,Y 353.302,Z 529.66,A -85,B 0,C 180,E1 12366.722,E2 12366.722} C_VEL
LIN {X 0,Y 353.245,Z 529.66,A -85,B 0,C 180,E1 12373.427,E2 12373.427} C_VEL
LIN {X 0,Y 353.293,Z 529.66,A -85,B 0,C 180,E1 12380.246,E2 12380.246} C_VEL
LIN {X 0,Y 353.416,Z 530.161,A -85,B 0,C 180,E1 12382.902,E2 12382.902} C_VEL
LIN {X 0,Y 372.982,Z 578.813,A -85,B 0,C 180,E1 12386.317,E2 12386.317} C_VEL
LIN {X 0,Y 377.162,Z 593.571,A -85,B 0,C 180,E1 12387.414,E2 12387.414} C_VEL
LIN {X 0,Y 373.095,Z 628.194,A -85,B 0,C 180,E1 12389.628,E2 12389.628} C_VEL
LIN {X 0,Y 368.261,Z 660.614,A -85,B 0,C 180,E1 12392.746,E2 12392.746} C_VEL
LIN {X 0,Y 363.773,Z 687.789,A -85,B 0,C 180,E1 12396.465,E2 12396.465} C_VEL
LIN {X 0,Y 359.865,Z 711.555,A -85,B 0,C 180,E1 12401.033,E2 12401.033} C_VEL
LIN {X 0,Y 357.234,Z 729.432,A -85,B 0,C 180,E1 12405.999,E2 12405.999} C_VEL
LIN {X 0,Y 355.856,Z 742.161,A -85,B 0,C 180,E1 12411.462,E2 12411.462} C_VEL
LIN {X 0,Y 355.43,Z 747.244,A -85,B 0,C 180,E1 12415.126,E2 12415.126} C_VEL
LIN {X 0,Y 355.321,Z 750.046,A -85,B 0,C 180,E1 12419.997,E2 12419.997} C_VEL
LIN {X 0,Y 355.532,Z 748.417,A -85,B 0,C 180,E1 12424.866,E2 12424.866} C_VEL
LIN {X 0,Y 356.425,Z 741.118,A -85,B 0,C 180,E1 12430.362,E2 12430.362} C_VEL
LIN {X 0,Y 358.304,Z 729.449,A -85,B 0,C 180,E1 12435.258,E2 12435.258} C_VEL
LIN {X 0,Y 361.791,Z 710.901,A -85,B 0,C 180,E1 12440.354,E2 12440.354} C_VEL
LIN {X 0,Y 366.712,Z 686.872,A -85,B 0,C 180,E1 12444.913,E2 12444.913} C_VEL
LIN {X 0,Y 372.506,Z 658.28,A -85,B 0,C 180,E1 12448.75,E2 12448.75} C_VEL
LIN {X 0,Y 378.57,Z 625.284,A -85,B 0,C 180,E1 12451.876,E2 12451.876} C_VEL
LIN {X 0,Y 383.364,Z 593.118,A -85,B 0,C 180,E1 12454.051,E2 12454.051} C_VEL
LIN {X 0,Y 379.555,Z 574.906,A -85,B 0,C 180,E1 12456.224,E2 12456.224} C_VEL
LIN {X 0,Y 374.76,Z 562.371,A -85,B 0,C 180,E1 12458.721,E2 12458.721} C_VEL
LIN {X 0,Y 372.558,Z 557.841,A -85,B 0,C 180,E1 12460.39,E2 12460.39} C_VEL
LIN {X 0,Y 371.412,Z 555.833,A -85,B 0,C 180,E1 12463.005,E2 12463.005} C_VEL
LIN {X 0,Y 373.789,Z 559.584,A -85,B 0,C 180,E1 12465.863,E2 12465.863} C_VEL
LIN {X 0,Y 378.501,Z 570.141,A -85,B 0,C 180,E1 12468.359,E2 12468.359} C_VEL
LIN {X 0,Y 383.219,Z 586.383,A -85,B 0,C 180,E1 12470.436,E2 12470.436} C_VEL
LIN {X 0,Y 384.735,Z 602.32,A -85,B 0,C 180,E1 12471.763,E2 12471.763} C_VEL
LIN {X 0,Y 378.557,Z 642.672,A -85,B 0,C 180,E1 12474.255,E2 12474.255} C_VEL
LIN {X 0,Y 372.388,Z 678.449,A -85,B 0,C 180,E1 12477.527,E2 12477.527} C_VEL
LIN {X 0,Y 366.557,Z 708.967,A -85,B 0,C 180,E1 12481.41,E2 12481.41} C_VEL
LIN {X 0,Y 361.621,Z 735.535,A -85,B 0,C 180,E1 12486.034,E2 12486.034} C_VEL
LIN {X 0,Y 358.005,Z 757.486,A -85,B 0,C 180,E1 12491.379,E2 12491.379} C_VEL
LIN {X 0,Y 356.036,Z 773.68,A -85,B 0,C 180,E1 12497.095,E2 12497.095} C_VEL
LIN {X 0,Y 355.345,Z 783.427,A -85,B 0,C 180,E1 12502.682,E2 12502.682} C_VEL
LIN {X 0,Y 355.198,Z 787.476,A -85,B 0,C 180,E1 12507.566,E2 12507.566} C_VEL
LIN {X 0,Y 355.206,Z 787.688,A -85,B 0,C 180,E1 12511.316,E2 12511.316} C_VEL
LIN {X 0,Y 352.705,Z 786.85,A -85,B 0,C 180,E1 12513.397,E2 12513.397} C_VEL
LIN {X 0,Y 347.477,Z 783.934,A -85,B 0,C 180,E1 12516.512,E2 12516.512} C_VEL
LIN {X 0,Y 347.403,Z 783.473,A -85,B 0,C 180,E1 12516.871,E2 12516.871} C_VEL
LIN {X 0,Y 348.009,Z 774.264,A -85,B 0,C 180,E1 12522.522,E2 12522.522} C_VEL
LIN {X 0,Y 349.731,Z 759.609,A -85,B 0,C 180,E1 12528.015,E2 12528.015} C_VEL
LIN {X 0,Y 352.842,Z 740.042,A -85,B 0,C 180,E1 12533.109,E2 12533.109} C_VEL
LIN {X 0,Y 357.643,Z 713.853,A -85,B 0,C 180,E1 12537.996,E2 12537.996} C_VEL
LIN {X 0,Y 363.136,Z 683.582,A -85,B 0,C 180,E1 12542.055,E2 12542.055} C_VEL
LIN {X 0,Y 368.756,Z 649.355,A -85,B 0,C 180,E1 12545.312,E2 12545.312} C_VEL
LIN {X 0,Y 373.696,Z 612.114,A -85,B 0,C 180,E1 12547.698,E2 12547.698} C_VEL
LIN {X 0,Y 374.228,Z 599.587,A -85,B 0,C 180,E1 12548.348,E2 12548.348} C_VEL
LIN {X 0,Y 358.307,Z 559.743,A -85,B 0,C 180,E1 12551.287,E2 12551.287} C_VEL
LIN {X 0,Y 345.34,Z 529.66,A -85,B 0,C 180,E1 12553.573,E2 12553.573} C_VEL
LIN {X 0,Y 345.24,Z 529.66,A -85,B 0,C 180,E1 12559.038,E2 12559.038} C_VEL
LIN {X 0,Y 345.443,Z 529.66,A -85,B 0,C 180,E1 12566.098,E2 12566.098} C_VEL
LIN {X 0,Y 345.679,Z 529.66,A -85,B 0,C 180,E1 12574.121,E2 12574.121} C_VEL
LIN {X 0,Y 345.981,Z 529.66,A -85,B 0,C 180,E1 12582.227,E2 12582.227} C_VEL
LIN {X 0,Y 346.36,Z 529.66,A -85,B 0,C 180,E1 12589.967,E2 12589.967} C_VEL
LIN {X 0,Y 347.039,Z 529.66,A -85,B 0,C 180,E1 12597.511,E2 12597.511} C_VEL
LIN {X 0,Y 346.784,Z 529.66,A -85,B 0,C 180,E1 12604.996,E2 12604.996} C_VEL
LIN {X 0,Y 346.377,Z 529.66,A -85,B 0,C 180,E1 12612.585,E2 12612.585} C_VEL
LIN {X 0,Y 345.913,Z 529.66,A -85,B 0,C 180,E1 12620.429,E2 12620.429} C_VEL
LIN {X 0,Y 345.656,Z 529.66,A -85,B 0,C 180,E1 12625.888,E2 12625.888} C_VEL
LIN {X 0,Y 345.372,Z 529.66,A -85,B 0,C 180,E1 12633.885,E2 12633.885} C_VEL
LIN {X 0,Y 345.444,Z 530.408,A -85,B 0,C 180,E1 12636.169,E2 12636.169} C_VEL
LIN {X 0,Y 362.055,Z 574.03,A -85,B 0,C 180,E1 12638.699,E2 12638.699} C_VEL
LIN {X 0,Y 363.617,Z 582.578,A -85,B 0,C 180,E1 12639.019,E2 12639.019} C_VEL
LIN {X 0,Y 362.088,Z 635.428,A -85,B 0,C 180,E1 12640.264,E2 12640.264} C_VEL
LIN {X 0,Y 359.787,Z 664.466,A -85,B 0,C 180,E1 12641.902,E2 12641.902} C_VEL
LIN {X 0,Y 356.788,Z 690.337,A -85,B 0,C 180,E1 12644.381,E2 12644.381} C_VEL
LIN {X 0,Y 353.493,Z 711.965,A -85,B 0,C 180,E1 12647.534,E2 12647.534} C_VEL
LIN {X 0,Y 350.613,Z 730.099,A -85,B 0,C 180,E1 12651.498,E2 12651.498} C_VEL
LIN {X 0,Y 348.804,Z 742.654,A -85,B 0,C 180,E1 12655.777,E2 12655.777} C_VEL
LIN {X 0,Y 347.662,Z 750.056,A -85,B 0,C 180,E1 12660.242,E2 12660.242} C_VEL
LIN {X 0,Y 346.993,Z 752.42,A -85,B 0,C 180,E1 12664.221,E2 12664.221} C_VEL
LIN {X 0,Y 347.337,Z 750.68,A -85,B 0,C 180,E1 12668.598,E2 12668.598} C_VEL
LIN {X 0,Y 348.368,Z 743.998,A -85,B 0,C 180,E1 12673.083,E2 12673.083} C_VEL
LIN {X 0,Y 350.058,Z 731.656,A -85,B 0,C 180,E1 12677.552,E2 12677.552} C_VEL
LIN {X 0,Y 352.631,Z 713.901,A -85,B 0,C 180,E1 12681.608,E2 12681.608} C_VEL
LIN {X 0,Y 355.775,Z 691.576,A -85,B 0,C 180,E1 12684.974,E2 12684.974} C_VEL
LIN {X 0,Y 358.86,Z 664.957,A -85,B 0,C 180,E1 12687.589,E2 12687.589} C_VEL
LIN {X 0,Y 361.046,Z 636.266,A -85,B 0,C 180,E1 12689.251,E2 12689.251} C_VEL
LIN {X 0,Y 362.215,Z 592.524,A -85,B 0,C 180,E1 12690.346,E2 12690.346} C_VEL
LIN {X 0,Y 361.789,Z 574.832,A -85,B 0,C 180,E1 12690.761,E2 12690.761} C_VEL
LIN {X 0,Y 347.726,Z 533,A -85,B 0,C 180,E1 12692.798,E2 12692.798} C_VEL
LIN {X 0,Y 346.952,Z 529.66,A -85,B 0,C 180,E1 12693.007,E2 12693.007} C_VEL
LIN {X 0,Y 346.39,Z 529.66,A -85,B 0,C 180,E1 12700.034,E2 12700.034} C_VEL
LIN {X 0,Y 345.984,Z 529.66,A -85,B 0,C 180,E1 12707.775,E2 12707.775} C_VEL
LIN {X 0,Y 345.648,Z 529.66,A -85,B 0,C 180,E1 12715.884,E2 12715.884} C_VEL
LIN {X 0,Y 345.402,Z 529.66,A -85,B 0,C 180,E1 12723.889,E2 12723.889} C_VEL
LIN {X 0,Y 345.254,Z 529.66,A -85,B 0,C 180,E1 12730.964,E2 12730.964} C_VEL
LIN {X 0,Y 345.246,Z 529.66,A -85,B 0,C 180,E1 12737.989,E2 12737.989} C_VEL
LIN {X 0,Y 345.407,Z 529.966,A -85,B 0,C 180,E1 12742.113,E2 12742.113} C_VEL
LIN {X 0,Y 365.289,Z 579.391,A -85,B 0,C 180,E1 12745.708,E2 12745.708} C_VEL
LIN {X 0,Y 369.996,Z 594.716,A -85,B 0,C 180,E1 12746.922,E2 12746.922} C_VEL
LIN {X 0,Y 365.633,Z 630.409,A -85,B 0,C 180,E1 12749.285,E2 12749.285} C_VEL
LIN {X 0,Y 360.834,Z 661.274,A -85,B 0,C 180,E1 12752.349,E2 12752.349} C_VEL
LIN {X 0,Y 355.987,Z 689.547,A -85,B 0,C 180,E1 12756.335,E2 12756.335} C_VEL
LIN {X 0,Y 352.029,Z 712.651,A -85,B 0,C 180,E1 12760.928,E2 12760.928} C_VEL
LIN {X 0,Y 349.301,Z 730.635,A -85,B 0,C 180,E1 12766.093,E2 12766.093} C_VEL
LIN {X 0,Y 348.004,Z 742.372,A -85,B 0,C 180,E1 12771.268,E2 12771.268} C_VEL
LIN {X 0,Y 347.416,Z 748.701,A -85,B 0,C 180,E1 12776.261,E2 12776.261} C_VEL
LIN {X 0,Y 347.432,Z 750.478,A -85,B 0,C 180,E1 12779.997,E2 12779.997} C_VEL
LIN {X 0,Y 347.685,Z 748.958,A -85,B 0,C 180,E1 12784.976,E2 12784.976} C_VEL
LIN {X 0,Y 348.661,Z 741.79,A -85,B 0,C 180,E1 12790.596,E2 12790.596} C_VEL
LIN {X 0,Y 350.691,Z 730.243,A -85,B 0,C 180,E1 12795.597,E2 12795.597} C_VEL
LIN {X 0,Y 354.23,Z 712.875,A -85,B 0,C 180,E1 12800.572,E2 12800.572} C_VEL
LIN {X 0,Y 359.325,Z 690.025,A -85,B 0,C 180,E1 12805.144,E2 12805.144} C_VEL
LIN {X 0,Y 365.545,Z 661.495,A -85,B 0,C 180,E1 12809.181,E2 12809.181} C_VEL
LIN {X 0,Y 372.162,Z 628.799,A -85,B 0,C 180,E1 12812.448,E2 12812.448} C_VEL
LIN {X 0,Y 377.884,Z 596.442,A -85,B 0,C 180,E1 12814.746,E2 12814.746} C_VEL
LIN {X 0,Y 375.139,Z 579.909,A -85,B 0,C 180,E1 12816.859,E2 12816.859} C_VEL
LIN {X 0,Y 371.542,Z 568.836,A -85,B 0,C 180,E1 12819.234,E2 12819.234} C_VEL
LIN {X 0,Y 369.804,Z 564.753,A -85,B 0,C 180,E1 12820.987,E2 12820.987} C_VEL
LIN {X 0,Y 369.443,Z 563.665,A -85,B 0,C 180,E1 12823.46,E2 12823.46} C_VEL
LIN {X 0,Y 371.183,Z 566.979,A -85,B 0,C 180,E1 12825.589,E2 12825.589} C_VEL
LIN {X 0,Y 375.173,Z 577.534,A -85,B 0,C 180,E1 12828.076,E2 12828.076} C_VEL
LIN {X 0,Y 378.71,Z 594.617,A -85,B 0,C 180,E1 12830.191,E2 12830.191} C_VEL
LIN {X 0,Y 378.815,Z 605.559,A -85,B 0,C 180,E1 12831.054,E2 12831.054} C_VEL
LIN {X 0,Y 371.85,Z 646.236,A -85,B 0,C 180,E1 12833.742,E2 12833.742} C_VEL
LIN {X 0,Y 365.112,Z 681.385,A -85,B 0,C 180,E1 12837.151,E2 12837.151} C_VEL
LIN {X 0,Y 359.079,Z 710.955,A -85,B 0,C 180,E1 12841.102,E2 12841.102} C_VEL
LIN {X 0,Y 353.758,Z 737.648,A -85,B 0,C 180,E1 12846.016,E2 12846.016} C_VEL
LIN {X 0,Y 350.038,Z 758.994,A -85,B 0,C 180,E1 12851.502,E2 12851.502} C_VEL
LIN {X 0,Y 348.187,Z 773.316,A -85,B 0,C 180,E1 12856.799,E2 12856.799} C_VEL
LIN {X 0,Y 347.469,Z 783.021,A -85,B 0,C 180,E1 12862.515,E2 12862.515} C_VEL
LIN {X 0,Y 347.317,Z 787.158,A -85,B 0,C 180,E1 12867.725,E2 12867.725} C_VEL
LIN {X 0,Y 347.387,Z 786.936,A -85,B 0,C 180,E1 12872.547,E2 12872.547} C_VEL
LIN {X 0,Y 347.403,Z 783.473,A -85,B 0,C 180,E1 12876.871,E2 12876.871} C_VEL
LIN {X 0,Y 345.069,Z 780.654,A -85,B 0,C 180,E1 12878.957,E2 12878.957} C_VEL
LIN {X 0,Y 340.102,Z 774.389,A -85,B 0,C 180,E1 12882.405,E2 12882.405} C_VEL
LIN {X 0,Y 341.805,Z 760.039,A -85,B 0,C 180,E1 12888.002,E2 12888.002} C_VEL
LIN {X 0,Y 345.047,Z 740.238,A -85,B 0,C 180,E1 12893.318,E2 12893.318} C_VEL
LIN {X 0,Y 349.997,Z 714.207,A -85,B 0,C 180,E1 12898.312,E2 12898.312} C_VEL
LIN {X 0,Y 355.609,Z 684.534,A -85,B 0,C 180,E1 12902.398,E2 12902.398} C_VEL
LIN {X 0,Y 361.474,Z 650.195,A -85,B 0,C 180,E1 12905.764,E2 12905.764} C_VEL
LIN {X 0,Y 366.417,Z 614.208,A -85,B 0,C 180,E1 12908.152,E2 12908.152} C_VEL
LIN {X 0,Y 367.03,Z 601.486,A -85,B 0,C 180,E1 12908.841,E2 12908.841} C_VEL
LIN {X 0,Y 351.089,Z 561.378,A -85,B 0,C 180,E1 12911.924,E2 12911.924} C_VEL
LIN {X 0,Y 337.362,Z 529.66,A -85,B 0,C 180,E1 12914.496,E2 12914.496} C_VEL
LIN {X 0,Y 337.317,Z 529.66,A -85,B 0,C 180,E1 12921.228,E2 12921.228} C_VEL
LIN {X 0,Y 337.526,Z 529.66,A -85,B 0,C 180,E1 12928.153,E2 12928.153} C_VEL
LIN {X 0,Y 337.835,Z 529.66,A -85,B 0,C 180,E1 12936.301,E2 12936.301} C_VEL
LIN {X 0,Y 338.016,Z 529.66,A -85,B 0,C 180,E1 12941.794,E2 12941.794} C_VEL
LIN {X 0,Y 338.42,Z 529.66,A -85,B 0,C 180,E1 12949.73,E2 12949.73} C_VEL
LIN {X 0,Y 339.12,Z 529.66,A -85,B 0,C 180,E1 12957.453,E2 12957.453} C_VEL
LIN {X 0,Y 339.04,Z 529.66,A -85,B 0,C 180,E1 12962.554,E2 12962.554} C_VEL
LIN {X 0,Y 338.498,Z 529.66,A -85,B 0,C 180,E1 12970.275,E2 12970.275} C_VEL
LIN {X 0,Y 338.093,Z 529.66,A -85,B 0,C 180,E1 12978.209,E2 12978.209} C_VEL
LIN {X 0,Y 337.823,Z 529.66,A -85,B 0,C 180,E1 12983.707,E2 12983.707} C_VEL
LIN {X 0,Y 337.495,Z 529.66,A -85,B 0,C 180,E1 12991.839,E2 12991.839} C_VEL
LIN {X 0,Y 337.486,Z 529.66,A -85,B 0,C 180,E1 12995.331,E2 12995.331} C_VEL
LIN {X 0,Y 355.06,Z 575.784,A -85,B 0,C 180,E1 12998.143,E2 12998.143} C_VEL
LIN {X 0,Y 356.542,Z 585.359,A -85,B 0,C 180,E1 12998.492,E2 12998.492} C_VEL
LIN {X 0,Y 354.936,Z 636.868,A -85,B 0,C 180,E1 12999.754,E2 12999.754} C_VEL
LIN {X 0,Y 352.441,Z 666.394,A -85,B 0,C 180,E1 13001.493,E2 13001.493} C_VEL
LIN {X 0,Y 349.263,Z 691.945,A -85,B 0,C 180,E1 13004.059,E2 13004.059} C_VEL
LIN {X 0,Y 345.595,Z 714.822,A -85,B 0,C 180,E1 13007.578,E2 13007.578} C_VEL
LIN {X 0,Y 342.803,Z 731.313,A -85,B 0,C 180,E1 13011.391,E2 13011.391} C_VEL
LIN {X 0,Y 341.016,Z 743.069,A -85,B 0,C 180,E1 13015.551,E2 13015.551} C_VEL
LIN {X 0,Y 339.967,Z 749.724,A -85,B 0,C 180,E1 13019.498,E2 13019.498} C_VEL
LIN {X 0,Y 339.143,Z 752.723,A -85,B 0,C 180,E1 13023.579,E2 13023.579} C_VEL
LIN {X 0,Y 339.111,Z 752.522,A -85,B 0,C 180,E1 13026.39,E2 13026.39} C_VEL
LIN {X 0,Y 340.044,Z 747.951,A -85,B 0,C 180,E1 13031.231,E2 13031.231} C_VEL
LIN {X 0,Y 341.497,Z 737.468,A -85,B 0,C 180,E1 13036.094,E2 13036.094} C_VEL
LIN {X 0,Y 343.973,Z 721.056,A -85,B 0,C 180,E1 13040.573,E2 13040.573} C_VEL
LIN {X 0,Y 346.997,Z 700.633,A -85,B 0,C 180,E1 13044.227,E2 13044.227} C_VEL
LIN {X 0,Y 350.324,Z 676.058,A -85,B 0,C 180,E1 13047.124,E2 13047.124} C_VEL
LIN {X 0,Y 352.929,Z 648.807,A -85,B 0,C 180,E1 13049.157,E2 13049.157} C_VEL
LIN {X 0,Y 354.523,Z 620.437,A -85,B 0,C 180,E1 13050.279,E2 13050.279} C_VEL
LIN {X 0,Y 354.72,Z 576.759,A -85,B 0,C 180,E1 13051.244,E2 13051.244} C_VEL
LIN {X 0,Y 340.373,Z 534.131,A -85,B 0,C 180,E1 13053.396,E2 13053.396} C_VEL
LIN {X 0,Y 338.982,Z 529.66,A -85,B 0,C 180,E1 13053.668,E2 13053.668} C_VEL
LIN {X 0,Y 338.367,Z 529.66,A -85,B 0,C 180,E1 13061.137,E2 13061.137} C_VEL
LIN {X 0,Y 338.016,Z 529.66,A -85,B 0,C 180,E1 13068.209,E2 13068.209} C_VEL
LIN {X 0,Y 337.812,Z 529.66,A -85,B 0,C 180,E1 13073.704,E2 13073.704} C_VEL
LIN {X 0,Y 337.506,Z 529.66,A -85,B 0,C 180,E1 13081.838,E2 13081.838} C_VEL
LIN {X 0,Y 337.332,Z 529.66,A -85,B 0,C 180,E1 13088.774,E2 13088.774} C_VEL
LIN {X 0,Y 337.337,Z 529.66,A -85,B 0,C 180,E1 13095.701,E2 13095.701} C_VEL
LIN {X 0,Y 337.388,Z 529.66,A -85,B 0,C 180,E1 13101.277,E2 13101.277} C_VEL
LIN {X 0,Y 357.645,Z 580.081,A -85,B 0,C 180,E1 13105.094,E2 13105.094} C_VEL
LIN {X 0,Y 362.691,Z 597.366,A -85,B 0,C 180,E1 13106.501,E2 13106.501} C_VEL
LIN {X 0,Y 358.18,Z 632.376,A -85,B 0,C 180,E1 13108.927,E2 13108.927} C_VEL
LIN {X 0,Y 352.9,Z 664.788,A -85,B 0,C 180,E1 13112.286,E2 13112.286} C_VEL
LIN {X 0,Y 348.115,Z 691.711,A -85,B 0,C 180,E1 13116.278,E2 13116.278} C_VEL
LIN {X 0,Y 343.987,Z 714.926,A -85,B 0,C 180,E1 13121.127,E2 13121.127} C_VEL
LIN {X 0,Y 341.318,Z 732.332,A -85,B 0,C 180,E1 13126.396,E2 13126.396} C_VEL
LIN {X 0,Y 340.022,Z 743.612,A -85,B 0,C 180,E1 13131.704,E2 13131.704} C_VEL
LIN {X 0,Y 339.5,Z 749.965,A -85,B 0,C 180,E1 13137.449,E2 13137.449} C_VEL
LIN {X 0,Y 339.684,Z 750.755,A -85,B 0,C 180,E1 13142.543,E2 13142.543} C_VEL
LIN {X 0,Y 340.131,Z 747.105,A -85,B 0,C 180,E1 13147.645,E2 13147.645} C_VEL
LIN {X 0,Y 341.546,Z 738.831,A -85,B 0,C 180,E1 13152.759,E2 13152.759} C_VEL
LIN {X 0,Y 344.502,Z 724.403,A -85,B 0,C 180,E1 13158.181,E2 13158.181} C_VEL
LIN {X 0,Y 349.157,Z 704.377,A -85,B 0,C 180,E1 13163.222,E2 13163.222} C_VEL
LIN {X 0,Y 355.489,Z 678.078,A -85,B 0,C 180,E1 13167.831,E2 13167.831} C_VEL
LIN {X 0,Y 362.794,Z 646.554,A -85,B 0,C 180,E1 13171.715,E2 13171.715} C_VEL
LIN {X 0,Y 370.379,Z 610.766,A -85,B 0,C 180,E1 13174.773,E2 13174.773} C_VEL
LIN {X 0,Y 372.461,Z 597.901,A -85,B 0,C 180,E1 13175.712,E2 13175.712} C_VEL
LIN {X 0,Y 370.431,Z 583.342,A -85,B 0,C 180,E1 13177.821,E2 13177.821} C_VEL
LIN {X 0,Y 367.949,Z 573.558,A -85,B 0,C 180,E1 13180.353,E2 13180.353} C_VEL
LIN {X 0,Y 367.1,Z 571.047,A -85,B 0,C 180,E1 13182.967,E2 13182.967} C_VEL
LIN {X 0,Y 368.539,Z 574.376,A -85,B 0,C 180,E1 13185.326,E2 13185.326} C_VEL
LIN {X 0,Y 371.489,Z 584.229,A -85,B 0,C 180,E1 13187.66,E2 13187.66} C_VEL
LIN {X 0,Y 373.635,Z 600.091,A -85,B 0,C 180,E1 13189.652,E2 13189.652} C_VEL
LIN {X 0,Y 373.091,Z 608.886,A -85,B 0,C 180,E1 13190.323,E2 13190.323} C_VEL
LIN {X 0,Y 365.577,Z 648.061,A -85,B 0,C 180,E1 13193.053,E2 13193.053} C_VEL
LIN {X 0,Y 358.19,Z 683.208,A -85,B 0,C 180,E1 13196.614,E2 13196.614} C_VEL
LIN {X 0,Y 351.628,Z 712.935,A -85,B 0,C 180,E1 13200.782,E2 13200.782} C_VEL
LIN {X 0,Y 346.024,Z 739.045,A -85,B 0,C 180,E1 13205.82,E2 13205.82} C_VEL
LIN {X 0,Y 342.118,Z 760.145,A -85,B 0,C 180,E1 13211.538,E2 13211.538} C_VEL
LIN {X 0,Y 340.164,Z 774.77,A -85,B 0,C 180,E1 13217.386,E2 13217.386} C_VEL
LIN {X 0,Y 339.576,Z 782.627,A -85,B 0,C 180,E1 13222.34,E2 13222.34} C_VEL
LIN {X 0,Y 339.432,Z 786.641,A -85,B 0,C 180,E1 13227.453,E2 13227.453} C_VEL
LIN {X 0,Y 339.514,Z 786.47,A -85,B 0,C 180,E1 13232.548,E2 13232.548} C_VEL
LIN {X 0,Y 339.571,Z 782.167,A -85,B 0,C 180,E1 13237.662,E2 13237.662} C_VEL
LIN {X 0,Y 340.102,Z 774.389,A -85,B 0,C 180,E1 13242.405,E2 13242.405} C_VEL
LIN {X 0,Y 336.716,Z 768.308,A -85,B 0,C 180,E1 13245.135,E2 13245.135} C_VEL
LIN {X 0,Y 333.804,Z 760.948,A -85,B 0,C 180,E1 13247.823,E2 13247.823} C_VEL
LIN {X 0,Y 337.174,Z 740.996,A -85,B 0,C 180,E1 13253.393,E2 13253.393} C_VEL
LIN {X 0,Y 342.022,Z 716.409,A -85,B 0,C 180,E1 13258.312,E2 13258.312} C_VEL
LIN {X 0,Y 347.727,Z 687.034,A -85,B 0,C 180,E1 13262.561,E2 13262.561} C_VEL
LIN {X 0,Y 353.758,Z 653.453,A -85,B 0,C 180,E1 13266.02,E2 13266.02} C_VEL
LIN {X 0,Y 359.212,Z 616.24,A -85,B 0,C 180,E1 13268.614,E2 13268.614} C_VEL
LIN {X 0,Y 359.869,Z 603.54,A -85,B 0,C 180,E1 13269.333,E2 13269.333} C_VEL
LIN {X 0,Y 344.855,Z 565.217,A -85,B 0,C 180,E1 13272.41,E2 13272.41} C_VEL
LIN {X 0,Y 329.447,Z 529.66,A -85,B 0,C 180,E1 13275.348,E2 13275.348} C_VEL
LIN {X 0,Y 329.398,Z 529.66,A -85,B 0,C 180,E1 13283.454,E2 13283.454} C_VEL
LIN {X 0,Y 329.647,Z 529.66,A -85,B 0,C 180,E1 13290.431,E2 13290.431} C_VEL
LIN {X 0,Y 329.945,Z 529.66,A -85,B 0,C 180,E1 13298.542,E2 13298.542} C_VEL
LIN {X 0,Y 330.359,Z 529.66,A -85,B 0,C 180,E1 13306.802,E2 13306.802} C_VEL
LIN {X 0,Y 330.914,Z 529.66,A -85,B 0,C 180,E1 13314.771,E2 13314.771} C_VEL
LIN {X 0,Y 331.287,Z 529.66,A -85,B 0,C 180,E1 13320.003,E2 13320.003} C_VEL
LIN {X 0,Y 330.726,Z 529.66,A -85,B 0,C 180,E1 13327.871,E2 13327.871} C_VEL
LIN {X 0,Y 330.291,Z 529.66,A -85,B 0,C 180,E1 13335.913,E2 13335.913} C_VEL
LIN {X 0,Y 329.817,Z 529.66,A -85,B 0,C 180,E1 13344.32,E2 13344.32} C_VEL
LIN {X 0,Y 329.544,Z 529.66,A -85,B 0,C 180,E1 13350.248,E2 13350.248} C_VEL
LIN {X 0,Y 329.548,Z 530.1,A -85,B 0,C 180,E1 13354.489,E2 13354.489} C_VEL
LIN {X 0,Y 347.165,Z 574.607,A -85,B 0,C 180,E1 13357.404,E2 13357.404} C_VEL
LIN {X 0,Y 349.621,Z 584.327,A -85,B 0,C 180,E1 13357.861,E2 13357.861} C_VEL
LIN {X 0,Y 347.935,Z 636.693,A -85,B 0,C 180,E1 13359.155,E2 13359.155} C_VEL
LIN {X 0,Y 345.401,Z 665.849,A -85,B 0,C 180,E1 13360.877,E2 13360.877} C_VEL
LIN {X 0,Y 342.09,Z 691.632,A -85,B 0,C 180,E1 13363.471,E2 13363.471} C_VEL
LIN {X 0,Y 338.292,Z 714.075,A -85,B 0,C 180,E1 13366.935,E2 13366.935} C_VEL
LIN {X 0,Y 335.236,Z 731.293,A -85,B 0,C 180,E1 13370.935,E2 13370.935} C_VEL
LIN {X 0,Y 333.065,Z 744.464,A -85,B 0,C 180,E1 13375.79,E2 13375.79} C_VEL
LIN {X 0,Y 331.946,Z 750.865,A -85,B 0,C 180,E1 13379.996,E2 13379.996} C_VEL
LIN {X 0,Y 331.338,Z 752.886,A -85,B 0,C 180,E1 13382.907,E2 13382.907} C_VEL
LIN {X 0,Y 331.193,Z 753.11,A -85,B 0,C 180,E1 13385.79,E2 13385.79} C_VEL
LIN {X 0,Y 331.858,Z 750.056,A -85,B 0,C 180,E1 13390.059,E2 13390.059} C_VEL
LIN {X 0,Y 333.237,Z 740.996,A -85,B 0,C 180,E1 13395.123,E2 13395.123} C_VEL
LIN {X 0,Y 335.41,Z 726.786,A -85,B 0,C 180,E1 13399.632,E2 13399.632} C_VEL
LIN {X 0,Y 338.523,Z 707.497,A -85,B 0,C 180,E1 13403.601,E2 13403.601} C_VEL
LIN {X 0,Y 342.07,Z 683.597,A -85,B 0,C 180,E1 13406.853,E2 13406.853} C_VEL
LIN {X 0,Y 345.053,Z 656.376,A -85,B 0,C 180,E1 13409.216,E2 13409.216} C_VEL
LIN {X 0,Y 347.04,Z 627.333,A -85,B 0,C 180,E1 13410.625,E2 13410.625} C_VEL
LIN {X 0,Y 347.473,Z 577.846,A -85,B 0,C 180,E1 13411.782,E2 13411.782} C_VEL
LIN {X 0,Y 333.778,Z 537.632,A -85,B 0,C 180,E1 13413.889,E2 13413.889} C_VEL
LIN {X 0,Y 331.006,Z 529.66,A -85,B 0,C 180,E1 13414.455,E2 13414.455} C_VEL
LIN {X 0,Y 330.532,Z 529.66,A -85,B 0,C 180,E1 13420.521,E2 13420.521} C_VEL
LIN {X 0,Y 330.07,Z 529.66,A -85,B 0,C 180,E1 13428.663,E2 13428.663} C_VEL
LIN {X 0,Y 329.803,Z 529.66,A -85,B 0,C 180,E1 13434.316,E2 13434.316} C_VEL
LIN {X 0,Y 329.573,Z 529.66,A -85,B 0,C 180,E1 13440.24,E2 13440.24} C_VEL
LIN {X 0,Y 329.432,Z 529.66,A -85,B 0,C 180,E1 13448.854,E2 13448.854} C_VEL
LIN {X 0,Y 329.415,Z 529.66,A -85,B 0,C 180,E1 13456.593,E2 13456.593} C_VEL
LIN {X 0,Y 329.444,Z 529.949,A -85,B 0,C 180,E1 13460.479,E2 13460.479} C_VEL
LIN {X 0,Y 349.42,Z 579.176,A -85,B 0,C 180,E1 13464.332,E2 13464.332} C_VEL
LIN {X 0,Y 355.46,Z 599.446,A -85,B 0,C 180,E1 13466.043,E2 13466.043} C_VEL
LIN {X 0,Y 350.674,Z 634.206,A -85,B 0,C 180,E1 13468.547,E2 13468.547} C_VEL
LIN {X 0,Y 345.304,Z 666.158,A -85,B 0,C 180,E1 13471.977,E2 13471.977} C_VEL
LIN {X 0,Y 340.197,Z 693.926,A -85,B 0,C 180,E1 13476.238,E2 13476.238} C_VEL
LIN {X 0,Y 336.19,Z 715.672,A -85,B 0,C 180,E1 13480.953,E2 13480.953} C_VEL
LIN {X 0,Y 333.454,Z 732.899,A -85,B 0,C 180,E1 13486.305,E2 13486.305} C_VEL
LIN {X 0,Y 332.046,Z 744.861,A -85,B 0,C 180,E1 13492.172,E2 13492.172} C_VEL
LIN {X 0,Y 331.617,Z 750.344,A -85,B 0,C 180,E1 13497.388,E2 13497.388} C_VEL
LIN {X 0,Y 331.823,Z 751.272,A -85,B 0,C 180,E1 13502.603,E2 13502.603} C_VEL
LIN {X 0,Y 332.298,Z 747.76,A -85,B 0,C 180,E1 13507.826,E2 13507.826} C_VEL
LIN {X 0,Y 334.158,Z 738.381,A -85,B 0,C 180,E1 13513.682,E2 13513.682} C_VEL
LIN {X 0,Y 337.457,Z 723.5,A -85,B 0,C 180,E1 13519.198,E2 13519.198} C_VEL
LIN {X 0,Y 342.844,Z 702.773,A -85,B 0,C 180,E1 13524.366,E2 13524.366} C_VEL
LIN {X 0,Y 349.816,Z 676.04,A -85,B 0,C 180,E1 13529.027,E2 13529.027} C_VEL
LIN {X 0,Y 357.933,Z 644.01,A -85,B 0,C 180,E1 13532.938,E2 13532.938} C_VEL
LIN {X 0,Y 366.597,Z 606.613,A -85,B 0,C 180,E1 13536.09,E2 13536.09} C_VEL
LIN {X 0,Y 367.462,Z 598.155,A -85,B 0,C 180,E1 13536.909,E2 13536.909} C_VEL
LIN {X 0,Y 365.967,Z 585.301,A -85,B 0,C 180,E1 13539.217,E2 13539.217} C_VEL
LIN {X 0,Y 364.792,Z 579.459,A -85,B 0,C 180,E1 13541.436,E2 13541.436} C_VEL
LIN {X 0,Y 364.911,Z 579.088,A -85,B 0,C 180,E1 13543.681,E2 13543.681} C_VEL
LIN {X 0,Y 366.133,Z 582.983,A -85,B 0,C 180,E1 13545.523,E2 13545.523} C_VEL
LIN {X 0,Y 367.97,Z 593.024,A -85,B 0,C 180,E1 13547.569,E2 13547.569} C_VEL
LIN {X 0,Y 368.585,Z 607.182,A -85,B 0,C 180,E1 13549.231,E2 13549.231} C_VEL
LIN {X 0,Y 359.817,Z 648.295,A -85,B 0,C 180,E1 13552.171,E2 13552.171} C_VEL
LIN {X 0,Y 351.639,Z 684.02,A -85,B 0,C 180,E1 13555.907,E2 13555.907} C_VEL
LIN {X 0,Y 344.205,Z 714.999,A -85,B 0,C 180,E1 13560.45,E2 13560.45} C_VEL
LIN {X 0,Y 338.307,Z 740.6,A -85,B 0,C 180,E1 13565.634,E2 13565.634} C_VEL
LIN {X 0,Y 334.266,Z 760.867,A -85,B 0,C 180,E1 13571.431,E2 13571.431} C_VEL
LIN {X 0,Y 332.273,Z 774.937,A -85,B 0,C 180,E1 13577.333,E2 13577.333} C_VEL
LIN {X 0,Y 331.63,Z 783.654,A -85,B 0,C 180,E1 13583.469,E2 13583.469} C_VEL
LIN {X 0,Y 331.559,Z 786.22,A -85,B 0,C 180,E1 13587.393,E2 13587.393} C_VEL
LIN {X 0,Y 331.642,Z 785.974,A -85,B 0,C 180,E1 13592.609,E2 13592.609} C_VEL
LIN {X 0,Y 331.699,Z 781.552,A -85,B 0,C 180,E1 13597.845,E2 13597.845} C_VEL
LIN {X 0,Y 332.316,Z 772.741,A -85,B 0,C 180,E1 13603.124,E2 13603.124} C_VEL
LIN {X 0,Y 333.804,Z 760.948,A -85,B 0,C 180,E1 13607.823,E2 13607.823} C_VEL
LIN {X 0,Y 331.251,Z 752.7,A -85,B 0,C 180,E1 13610.444,E2 13610.444} C_VEL
LIN {X 0,Y 328.996,Z 743.52,A -85,B 0,C 180,E1 13613.03,E2 13613.03} C_VEL
LIN {X 0,Y 333.967,Z 718.78,A -85,B 0,C 180,E1 13618.253,E2 13618.253} C_VEL
LIN {X 0,Y 340.001,Z 688.905,A -85,B 0,C 180,E1 13622.792,E2 13622.792} C_VEL
LIN {X 0,Y 346.246,Z 655.328,A -85,B 0,C 180,E1 13626.384,E2 13626.384} C_VEL
LIN {X 0,Y 352.041,Z 617.92,A -85,B 0,C 180,E1 13629.103,E2 13629.103} C_VEL
LIN {X 0,Y 353.129,Z 606.818,A -85,B 0,C 180,E1 13629.726,E2 13629.726} C_VEL
LIN {X 0,Y 338.556,Z 568.948,A -85,B 0,C 180,E1 13632.898,E2 13632.898} C_VEL
LIN {X 0,Y 321.527,Z 529.66,A -85,B 0,C 180,E1 13636.197,E2 13636.197} C_VEL
LIN {X 0,Y 321.471,Z 529.66,A -85,B 0,C 180,E1 13642.94,E2 13642.94} C_VEL
LIN {X 0,Y 321.557,Z 529.66,A -85,B 0,C 180,E1 13648.927,E2 13648.927} C_VEL
LIN {X 0,Y 321.823,Z 529.66,A -85,B 0,C 180,E1 13655.043,E2 13655.043} C_VEL
LIN {X 0,Y 322.093,Z 529.66,A -85,B 0,C 180,E1 13660.86,E2 13660.86} C_VEL
LIN {X 0,Y 322.588,Z 529.66,A -85,B 0,C 180,E1 13669.22,E2 13669.22} C_VEL
LIN {X 0,Y 323.279,Z 529.66,A -85,B 0,C 180,E1 13677.328,E2 13677.328} C_VEL
LIN {X 0,Y 323.219,Z 529.66,A -85,B 0,C 180,E1 13682.679,E2 13682.679} C_VEL
LIN {X 0,Y 322.66,Z 529.66,A -85,B 0,C 180,E1 13690.847,E2 13690.847} C_VEL
LIN {X 0,Y 322.147,Z 529.66,A -85,B 0,C 180,E1 13699.144,E2 13699.144} C_VEL
LIN {X 0,Y 321.755,Z 529.66,A -85,B 0,C 180,E1 13706.989,E2 13706.989} C_VEL
LIN {X 0,Y 321.658,Z 529.688,A -85,B 0,C 180,E1 13713.563,E2 13713.563} C_VEL
LIN {X 0,Y 339.563,Z 574.449,A -85,B 0,C 180,E1 13716.675,E2 13716.675} C_VEL
LIN {X 0,Y 342.673,Z 584.686,A -85,B 0,C 180,E1 13717.226,E2 13717.226} C_VEL
LIN {X 0,Y 340.93,Z 637.257,A -85,B 0,C 180,E1 13718.557,E2 13718.557} C_VEL
LIN {X 0,Y 338.257,Z 666.66,A -85,B 0,C 180,E1 13720.339,E2 13720.339} C_VEL
LIN {X 0,Y 334.674,Z 692.893,A -85,B 0,C 180,E1 13723.064,E2 13723.064} C_VEL
LIN {X 0,Y 330.841,Z 714.365,A -85,B 0,C 180,E1 13726.462,E2 13726.462} C_VEL
LIN {X 0,Y 327.719,Z 731.041,A -85,B 0,C 180,E1 13730.384,E2 13730.384} C_VEL
LIN {X 0,Y 325.469,Z 743.626,A -85,B 0,C 180,E1 13734.935,E2 13734.935} C_VEL
LIN {X 0,Y 324.25,Z 750.54,A -85,B 0,C 180,E1 13739.207,E2 13739.207} C_VEL
LIN {X 0,Y 323.537,Z 753.121,A -85,B 0,C 180,E1 13742.402,E2 13742.402} C_VEL
LIN {X 0,Y 323.282,Z 753.589,A -85,B 0,C 180,E1 13745.158,E2 13745.158} C_VEL
LIN {X 0,Y 323.935,Z 750.745,A -85,B 0,C 180,E1 13749.89,E2 13749.89} C_VEL
LIN {X 0,Y 325.186,Z 743.212,A -85,B 0,C 180,E1 13754.524,E2 13754.524} C_VEL
LIN {X 0,Y 327.375,Z 729.307,A -85,B 0,C 180,E1 13759.374,E2 13759.374} C_VEL
LIN {X 0,Y 330.511,Z 711.062,A -85,B 0,C 180,E1 13763.445,E2 13763.445} C_VEL
LIN {X 0,Y 334.084,Z 688.354,A -85,B 0,C 180,E1 13766.809,E2 13766.809} C_VEL
LIN {X 0,Y 337.285,Z 661.987,A -85,B 0,C 180,E1 13769.358,E2 13769.358} C_VEL
LIN {X 0,Y 339.585,Z 634.255,A -85,B 0,C 180,E1 13770.926,E2 13770.926} C_VEL
LIN {X 0,Y 340.458,Z 579.787,A -85,B 0,C 180,E1 13772.301,E2 13772.301} C_VEL
LIN {X 0,Y 326.927,Z 540.361,A -85,B 0,C 180,E1 13774.442,E2 13774.442} C_VEL
LIN {X 0,Y 323.054,Z 529.66,A -85,B 0,C 180,E1 13775.118,E2 13775.118} C_VEL
LIN {X 0,Y 322.431,Z 529.66,A -85,B 0,C 180,E1 13783.532,E2 13783.532} C_VEL
LIN {X 0,Y 321.993,Z 529.66,A -85,B 0,C 180,E1 13792.018,E2 13792.018} C_VEL
LIN {X 0,Y 321.711,Z 529.66,A -85,B 0,C 180,E1 13797.971,E2 13797.971} C_VEL
LIN {X 0,Y 321.482,Z 529.66,A -85,B 0,C 180,E1 13804.28,E2 13804.28} C_VEL
LIN {X 0,Y 321.405,Z 529.66,A -85,B 0,C 180,E1 13811.301,E2 13811.301} C_VEL
LIN {X 0,Y 321.46,Z 529.66,A -85,B 0,C 180,E1 13819.544,E2 13819.544} C_VEL
LIN {X 0,Y 341.923,Z 580.275,A -85,B 0,C 180,E1 13823.715,E2 13823.715} C_VEL
LIN {X 0,Y 348.32,Z 600.411,A -85,B 0,C 180,E1 13825.511,E2 13825.511} C_VEL
LIN {X 0,Y 343.503,Z 634.187,A -85,B 0,C 180,E1 13827.998,E2 13827.998} C_VEL
LIN {X 0,Y 337.95,Z 666.245,A -85,B 0,C 180,E1 13831.493,E2 13831.493} C_VEL
LIN {X 0,Y 332.593,Z 694.402,A -85,B 0,C 180,E1 13835.896,E2 13835.896} C_VEL
LIN {X 0,Y 328.338,Z 716.7,A -85,B 0,C 180,E1 13840.855,E2 13840.855} C_VEL
LIN {X 0,Y 325.701,Z 732.719,A -85,B 0,C 180,E1 13845.919,E2 13845.919} C_VEL
LIN {X 0,Y 324.359,Z 743.943,A -85,B 0,C 180,E1 13851.3,E2 13851.3} C_VEL
LIN {X 0,Y 323.726,Z 750.706,A -85,B 0,C 180,E1 13857.325,E2 13857.325} C_VEL
LIN {X 0,Y 323.939,Z 751.8,A -85,B 0,C 180,E1 13862.666,E2 13862.666} C_VEL
LIN {X 0,Y 324.481,Z 748.441,A -85,B 0,C 180,E1 13868.016,E2 13868.016} C_VEL
LIN {X 0,Y 326.44,Z 739.458,A -85,B 0,C 180,E1 13873.899,E2 13873.899} C_VEL
LIN {X 0,Y 330.133,Z 724.3,A -85,B 0,C 180,E1 13879.759,E2 13879.759} C_VEL
LIN {X 0,Y 336.231,Z 702.845,A -85,B 0,C 180,E1 13885.232,E2 13885.232} C_VEL
LIN {X 0,Y 343.806,Z 676.322,A -85,B 0,C 180,E1 13889.947,E2 13889.947} C_VEL
LIN {X 0,Y 352.798,Z 644.076,A -85,B 0,C 180,E1 13893.962,E2 13893.962} C_VEL
LIN {X 0,Y 362.439,Z 606.978,A -85,B 0,C 180,E1 13897.167,E2 13897.167} C_VEL
LIN {X 0,Y 362.837,Z 596.894,A -85,B 0,C 180,E1 13898.592,E2 13898.592} C_VEL
LIN {X 0,Y 362.256,Z 588.192,A -85,B 0,C 180,E1 13900.84,E2 13900.84} C_VEL
LIN {X 0,Y 362.084,Z 586.597,A -85,B 0,C 180,E1 13901.816,E2 13901.816} C_VEL
LIN {X 0,Y 362.679,Z 587.788,A -85,B 0,C 180,E1 13904.424,E2 13904.424} C_VEL
LIN {X 0,Y 363.698,Z 596.367,A -85,B 0,C 180,E1 13906.577,E2 13906.577} C_VEL
LIN {X 0,Y 363.765,Z 609.268,A -85,B 0,C 180,E1 13908.299,E2 13908.299} C_VEL
LIN {X 0,Y 353.856,Z 650.613,A -85,B 0,C 180,E1 13911.417,E2 13911.417} C_VEL
LIN {X 0,Y 344.844,Z 686.21,A -85,B 0,C 180,E1 13915.33,E2 13915.33} C_VEL
LIN {X 0,Y 337.267,Z 715.377,A -85,B 0,C 180,E1 13919.78,E2 13919.78} C_VEL
LIN {X 0,Y 330.985,Z 740.595,A -85,B 0,C 180,E1 13925.058,E2 13925.058} C_VEL
LIN {X 0,Y 326.531,Z 761.093,A -85,B 0,C 180,E1 13931.127,E2 13931.127} C_VEL
LIN {X 0,Y 324.404,Z 775.085,A -85,B 0,C 180,E1 13937.25,E2 13937.25} C_VEL
LIN {X 0,Y 323.743,Z 783.283,A -85,B 0,C 180,E1 13943.309,E2 13943.309} C_VEL
LIN {X 0,Y 323.661,Z 785.781,A -85,B 0,C 180,E1 13947.329,E2 13947.329} C_VEL
LIN {X 0,Y 323.745,Z 785.468,A -85,B 0,C 180,E1 13952.673,E2 13952.673} C_VEL
LIN {X 0,Y 323.82,Z 780.914,A -85,B 0,C 180,E1 13958.037,E2 13958.037} C_VEL
LIN {X 0,Y 324.501,Z 771.93,A -85,B 0,C 180,E1 13963.446,E2 13963.446} C_VEL
LIN {X 0,Y 326.526,Z 756.975,A -85,B 0,C 180,E1 13969.226,E2 13969.226} C_VEL
LIN {X 0,Y 328.996,Z 743.52,A -85,B 0,C 180,E1 13973.03,E2 13973.03} C_VEL
LIN {X 0,Y 327.054,Z 733.541,A -85,B 0,C 180,E1 13975.527,E2 13975.527} C_VEL
LIN {X 0,Y 325.518,Z 722.568,A -85,B 0,C 180,E1 13977.919,E2 13977.919} C_VEL
LIN {X 0,Y 331.659,Z 693.315,A -85,B 0,C 180,E1 13982.66,E2 13982.66} C_VEL
LIN {X 0,Y 338.117,Z 660.308,A -85,B 0,C 180,E1 13986.471,E2 13986.471} C_VEL
LIN {X 0,Y 344.223,Z 623.333,A -85,B 0,C 180,E1 13989.371,E2 13989.371} C_VEL
LIN {X 0,Y 345.734,Z 608.302,A -85,B 0,C 180,E1 13990.285,E2 13990.285} C_VEL
LIN {X 0,Y 331.175,Z 570.212,A -85,B 0,C 180,E1 13993.596,E2 13993.596} C_VEL
LIN {X 0,Y 313.591,Z 529.66,A -85,B 0,C 180,E1 13997.204,E2 13997.204} C_VEL
LIN {X 0,Y 313.539,Z 529.66,A -85,B 0,C 180,E1 14004.904,E2 14004.904} C_VEL
LIN {X 0,Y 313.704,Z 529.66,A -85,B 0,C 180,E1 14011.252,E2 14011.252} C_VEL
LIN {X 0,Y 313.998,Z 529.66,A -85,B 0,C 180,E1 14017.394,E2 14017.394} C_VEL
